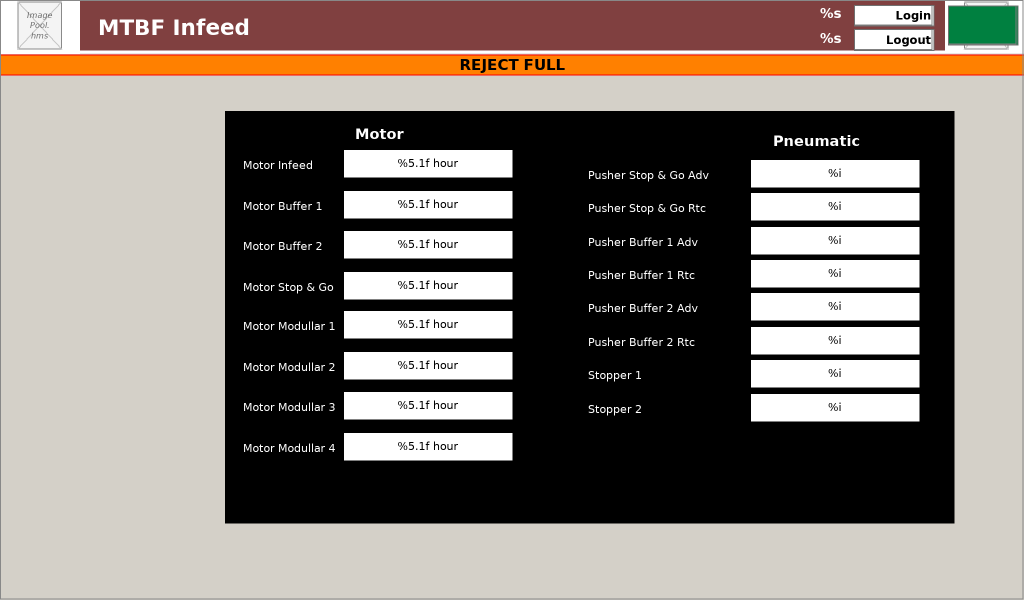
VISUALIZATION MTBF_Infeed  // 1024x600
    Frame (0,-2 1021x55)
        shows Header()
    Label (95,15 250x25), "MTBF Infeed"
    RoundedRectangle (225,111 729x412)
    Label (243,114 273x40), "Motor"
    Label (240,148 103x35), "Motor Infeed"
    RoundedRectangle (343,149 170x29), "%5.1f hour", text variable: InputOutput_GVL.MTBF_Motor[8]
    Label (240,189 103x35), "Motor Buffer 1"
    RoundedRectangle (343,190 170x29), "%5.1f hour", text variable: InputOutput_GVL.MTBF_Motor[9]
    Label (240,229 103x35), "Motor Buffer 2"
    RoundedRectangle (343,230 170x29), "%5.1f hour", text variable: InputOutput_GVL.MTBF_Motor[10]
    Label (240,270 103x35), "Motor Stop & Go"
    RoundedRectangle (343,271 170x29), "%5.1f hour", text variable: InputOutput_GVL.MTBF_Motor[11]
    Label (240,309 103x35), "Motor Modullar 1"
    RoundedRectangle (343,310 170x29), "%5.1f hour", text variable: InputOutput_GVL.MTBF_Motor[12]
    Label (240,350 103x35), "Motor Modullar 2"
    RoundedRectangle (343,351 170x29), "%5.1f hour", text variable: InputOutput_GVL.MTBF_Motor[13]
    Label (240,390 103x35), "Motor Modullar 3"
    RoundedRectangle (343,391 170x29), "%5.1f hour", text variable: InputOutput_GVL.MTBF_Motor[14]
    Label (240,431 103x35), "Motor Modullar 4"
    RoundedRectangle (343,432 170x29), "%5.1f hour", text variable: InputOutput_GVL.MTBF_Motor[15]
    Label (585,158 147x35), "Pusher Stop & Go Adv"
    RoundedRectangle (750,159 170x29), "%i", text variable: InputOutput_GVL.MTBF_Pneumatic[1]
    Label (680,121 273x40), "Pneumatic"
    Label (585,191 147x35), "Pusher Stop & Go Rtc"
    RoundedRectangle (750,192 170x29), "%i", text variable: InputOutput_GVL.MTBF_Pneumatic[2]
    Label (585,225 147x35), "Pusher Buffer 1 Adv"
    RoundedRectangle (750,226 170x29), "%i", text variable: InputOutput_GVL.MTBF_Pneumatic[3]
    Label (585,258 147x35), "Pusher Buffer 1 Rtc"
    RoundedRectangle (750,259 170x29), "%i", text variable: InputOutput_GVL.MTBF_Pneumatic[4]
    Label (585,291 147x35), "Pusher Buffer 2 Adv"
    RoundedRectangle (750,292 170x29), "%i", text variable: InputOutput_GVL.MTBF_Pneumatic[5]
    Label (585,325 147x35), "Pusher Buffer 2 Rtc"
    RoundedRectangle (750,326 170x29), "%i", text variable: InputOutput_GVL.MTBF_Pneumatic[6]
    Label (585,358 147x35), "Stopper 1"
    RoundedRectangle (750,359 170x29), "%i", text variable: InputOutput_GVL.MTBF_Pneumatic[7]
    Label (585,392 147x35), "Stopper 2"
    RoundedRectangle (750,393 170x29), "%i", text variable: InputOutput_GVL.MTBF_Pneumatic[8]
END_VISUALIZATION

// ---- VISUs/MTBF/MTBF_Shuttle.TcVIS
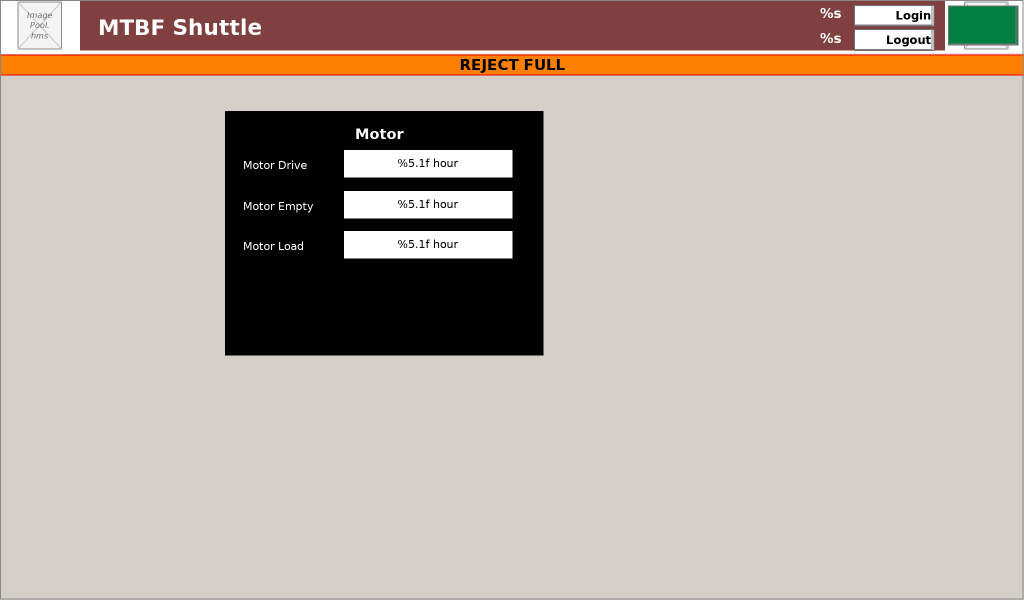
VISUALIZATION MTBF_Shuttle  // 1024x600
    Frame (0,-2 1021x55)
        shows Header()
    Label (95,15 250x25), "MTBF Shuttle"
    RoundedRectangle (225,111 318x244)
    Label (243,114 273x40), "Motor"
    Label (240,148 103x35), "Motor Drive"
    RoundedRectangle (343,149 170x29), "%5.1f hour", text variable: InputOutput_GVL.MTBF_Motor[16]
    Label (240,189 103x35), "Motor Empty"
    RoundedRectangle (343,190 170x29), "%5.1f hour", text variable: InputOutput_GVL.MTBF_Motor[17]
    Label (240,229 103x35), "Motor Load"
    RoundedRectangle (343,230 170x29), "%5.1f hour", text variable: InputOutput_GVL.MTBF_Motor[18]
END_VISUALIZATION

// ---- VISUs/MTBF/MTBF_Dispenser.TcVIS
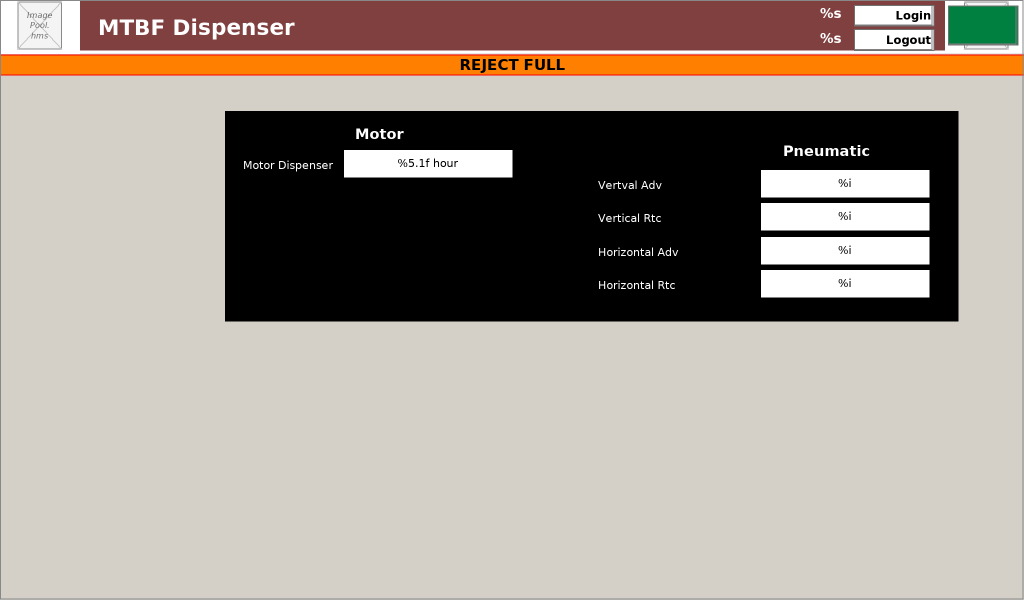
VISUALIZATION MTBF_Dispenser  // 1024x600
    Frame (0,-2 1021x55)
        shows Header()
    Label (95,15 250x25), "MTBF Dispenser"
    RoundedRectangle (225,111 733x210)
    Label (243,114 273x40), "Motor"
    Label (240,148 103x35), "Motor Dispenser"
    RoundedRectangle (343,149 170x29), "%5.1f hour", text variable: InputOutput_GVL.MTBF_Motor[19]
    Label (595,168 147x35), "Vertval Adv"
    RoundedRectangle (760,169 170x29), "%i", text variable: InputOutput_GVL.MTBF_Pneumatic[9]
    Label (690,131 273x40), "Pneumatic"
    Label (595,201 147x35), "Vertical Rtc"
    RoundedRectangle (760,202 170x29), "%i", text variable: InputOutput_GVL.MTBF_Pneumatic[10]
    Label (595,235 147x35), "Horizontal Adv"
    RoundedRectangle (760,236 170x29), "%i", text variable: InputOutput_GVL.MTBF_Pneumatic[11]
    Label (595,268 147x35), "Horizontal Rtc"
    RoundedRectangle (760,269 170x29), "%i", text variable: InputOutput_GVL.MTBF_Pneumatic[12]
END_VISUALIZATION

// ---- VISUs/OEE/OEE.TcVIS
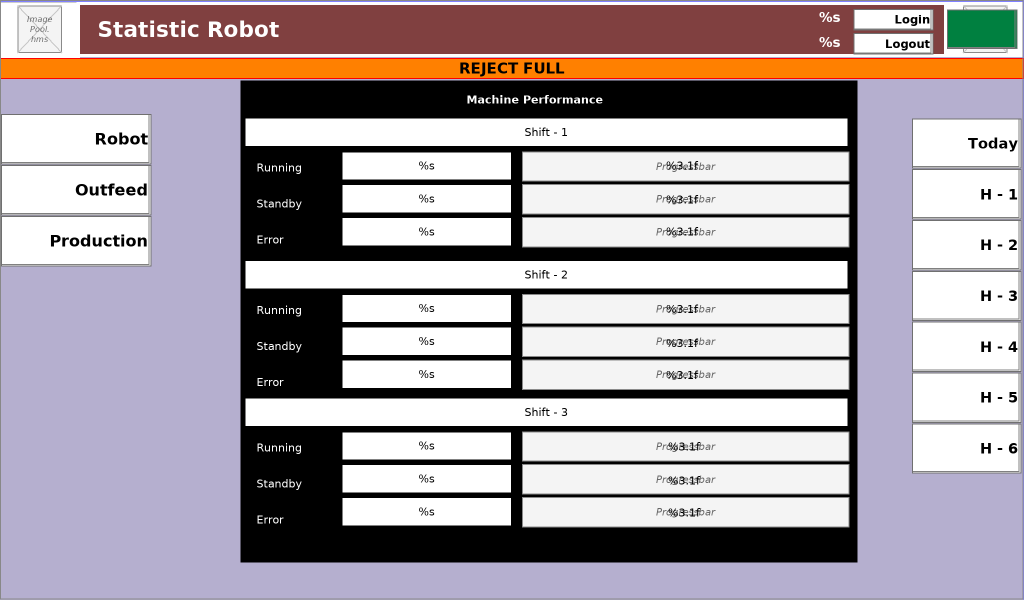
VISUALIZATION OEE  // 1024x600
    Frame (0,2 1023x598)
        shows OEE_Robot()
        shows OEE_Outfeed()
        shows OEE_Counter()
        shows Test_Place1()
        shows Test_Place2()
        shows Test_Place3()
        shows Test_Place4()
    Button (1,114 150x50), "Robot", image: VisuSymbols.Symbols.Database2
        OnMouseDown: FrameSelectionChange Selection=SelectedFrame=146e207b-fd78-4676-ba16-384fa245d7d2, GlobSel=AssignDir=MainPage.GenElemInst_1003, AssignType=Directly, SelType=Locally
    Button (1,165 150x50), "Outfeed", image: VisuSymbols.Symbols.Database2
        OnMouseDown: FrameSelectionChange Selection=SelectedFrame=146e207b-fd78-4676-ba16-384fa245d7d2, Selection=1, GlobSel=AssignDir=MainPage.GenElemInst_1003, AssignType=Directly, SelType=Locally
    Button (1,216 150x50), "Production", image: VisuSymbols.Symbols.Database2
        OnMouseDown: FrameSelectionChange Selection=SelectedFrame=146e207b-fd78-4676-ba16-384fa245d7d2, Selection=2, GlobSel=AssignDir=MainPage.GenElemInst_1003, AssignType=Directly, SelType=Locally
END_VISUALIZATION

// ---- VISUs/OEE/OEE_Outfeed.TcVIS
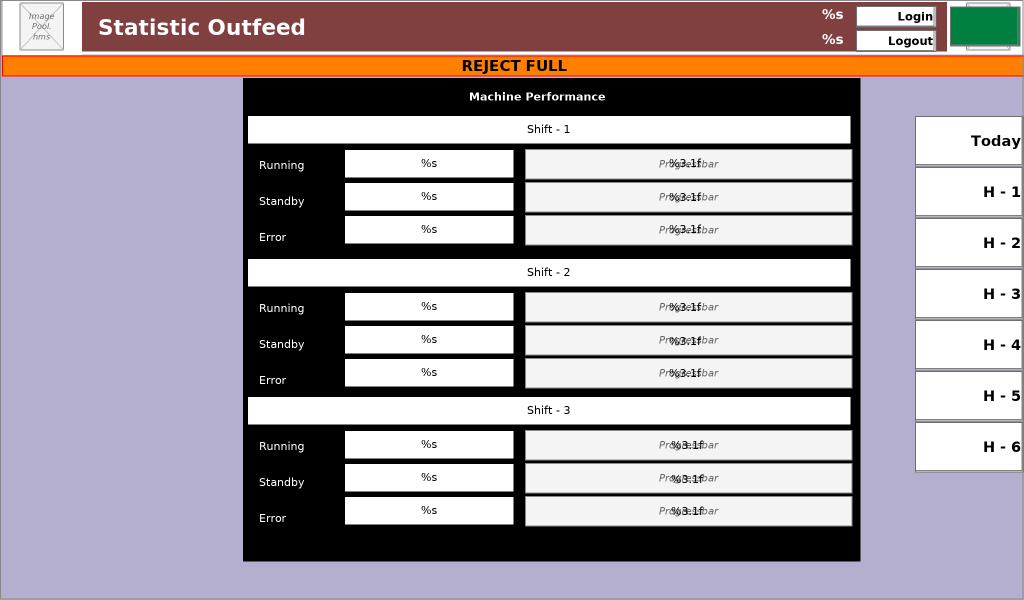
VISUALIZATION OEE_Outfeed  // 1024x600
    Frame (2,-1 1021x55)
        shows Header()
    RoundedRectangle (243,78 617x483)
    RoundedRectangle (247,115 604x29), "Shift - 1"
    Label (270,77 535x40), "Machine Performance"
    Label (256,148 78x35), "Running"
    Label (256,184 78x35), "Standby"
    Label (256,220 78x35), "Error"
    Progressbar (525,149 327x30), variable: Data_GVL.dt_OEEOutfeed.Precentage[0].Running
    Progressbar (525,182 327x30), variable: Data_GVL.dt_OEEOutfeed.Precentage[0].Stopped
    Progressbar (525,215 327x30), variable: Data_GVL.dt_OEEOutfeed.Precentage[0].Error
    RoundedRectangle (344,149 170x29), "%s", text variable: Data_GVL.dt_OEEOutfeed.HMI_Time[0].sRunning
    RoundedRectangle (344,182 170x29), "%s", text variable: Data_GVL.dt_OEEOutfeed.HMI_Time[0].sStopped
    RoundedRectangle (344,215 170x29), "%s", text variable: Data_GVL.dt_OEEOutfeed.HMI_Time[0].sError
    RoundedRectangle (247,258 604x29), "Shift - 2"
    Label (256,291 78x35), "Running"
    Label (256,327 78x35), "Standby"
    Label (256,363 78x35), "Error"
    Progressbar (525,292 327x30), variable: Data_GVL.dt_OEEOutfeed.Precentage[1].Running
    Progressbar (525,325 327x30), variable: Data_GVL.dt_OEEOutfeed.Precentage[1].Stopped
    Progressbar (525,358 327x30), variable: Data_GVL.dt_OEEOutfeed.Precentage[1].Error
    RoundedRectangle (344,292 170x29), "%s", text variable: Data_GVL.dt_OEEOutfeed.HMI_Time[1].sRunning
    RoundedRectangle (344,325 170x29), "%s", text variable: Data_GVL.dt_OEEOutfeed.HMI_Time[1].sStopped
    RoundedRectangle (344,358 170x29), "%s", text variable: Data_GVL.dt_OEEOutfeed.HMI_Time[1].sError
    RoundedRectangle (247,396 604x29), "Shift - 3"
    Label (256,429 78x35), "Running"
    Label (256,465 78x35), "Standby"
    Label (256,501 78x35), "Error"
    Progressbar (525,430 327x30), variable: Data_GVL.dt_OEEOutfeed.Precentage[2].Running
    Progressbar (525,463 327x30), variable: Data_GVL.dt_OEEOutfeed.Precentage[2].Stopped
    Progressbar (525,496 327x30), variable: Data_GVL.dt_OEEOutfeed.Precentage[2].Error
    RoundedRectangle (344,430 170x29), "%s", text variable: Data_GVL.dt_OEEOutfeed.HMI_Time[2].sRunning
    RoundedRectangle (344,463 170x29), "%s", text variable: Data_GVL.dt_OEEOutfeed.HMI_Time[2].sStopped
    RoundedRectangle (344,496 170x29), "%s", text variable: Data_GVL.dt_OEEOutfeed.HMI_Time[2].sError
    Button (915,116 109x50), "Today", image: VisuSymbols.Symbols.CalenderDay
        OnMouseClick: execute { Data_GVL.dt_OEEOutfeed.HMI_NumberPrev := 0; }
    Button (915,167 109x50), "H - 1", image: VisuSymbols.Symbols.CalenderDay
        OnMouseClick: execute { Data_GVL.dt_OEEOutfeed.HMI_NumberPrev := 1; }
    Button (915,218 109x50), "H - 2", image: VisuSymbols.Symbols.CalenderDay
        OnMouseClick: execute { Data_GVL.dt_OEEOutfeed.HMI_NumberPrev := 2; }
    Button (915,269 109x50), "H - 3", image: VisuSymbols.Symbols.CalenderDay
        OnMouseClick: execute { Data_GVL.dt_OEEOutfeed.HMI_NumberPrev := 3; }
    Button (915,320 109x50), "H - 4", image: VisuSymbols.Symbols.CalenderDay
        OnMouseClick: execute { Data_GVL.dt_OEEOutfeed.HMI_NumberPrev := 4; }
    Button (915,371 109x50), "H - 5", image: VisuSymbols.Symbols.CalenderDay
        OnMouseClick: execute { Data_GVL.dt_OEEOutfeed.HMI_NumberPrev := 5; }
    Button (915,422 109x50), "H - 6", image: VisuSymbols.Symbols.CalenderDay
        OnMouseClick: execute { Data_GVL.dt_OEEOutfeed.HMI_NumberPrev := 6; }
    RoundedRectangle (600,149 170x29), "%3.1f", text variable: Data_GVL.dt_OEEOutfeed.Precentage[0].Running
    RoundedRectangle (600,183 170x29), "%3.1f", text variable: Data_GVL.dt_OEEOutfeed.Precentage[0].Stopped
    RoundedRectangle (600,215 170x29), "%3.1f", text variable: Data_GVL.dt_OEEOutfeed.Precentage[0].Error
    RoundedRectangle (600,293 170x29), "%3.1f", text variable: Data_GVL.dt_OEEOutfeed.Precentage[1].Running
    RoundedRectangle (600,327 170x29), "%3.1f", text variable: Data_GVL.dt_OEEOutfeed.Precentage[1].Stopped
    RoundedRectangle (600,359 170x29), "%3.1f", text variable: Data_GVL.dt_OEEOutfeed.Precentage[1].Error
    RoundedRectangle (602,431 170x29), "%3.1f", text variable: Data_GVL.dt_OEEOutfeed.Precentage[2].Running
    RoundedRectangle (602,465 170x29), "%3.1f", text variable: Data_GVL.dt_OEEOutfeed.Precentage[2].Stopped
    RoundedRectangle (602,497 170x29), "%3.1f", text variable: Data_GVL.dt_OEEOutfeed.Precentage[2].Error
    Label (95,15 214x25), "Statistic Outfeed"
END_VISUALIZATION

// ---- VISUs/OEE/OEE_Robot.TcVIS
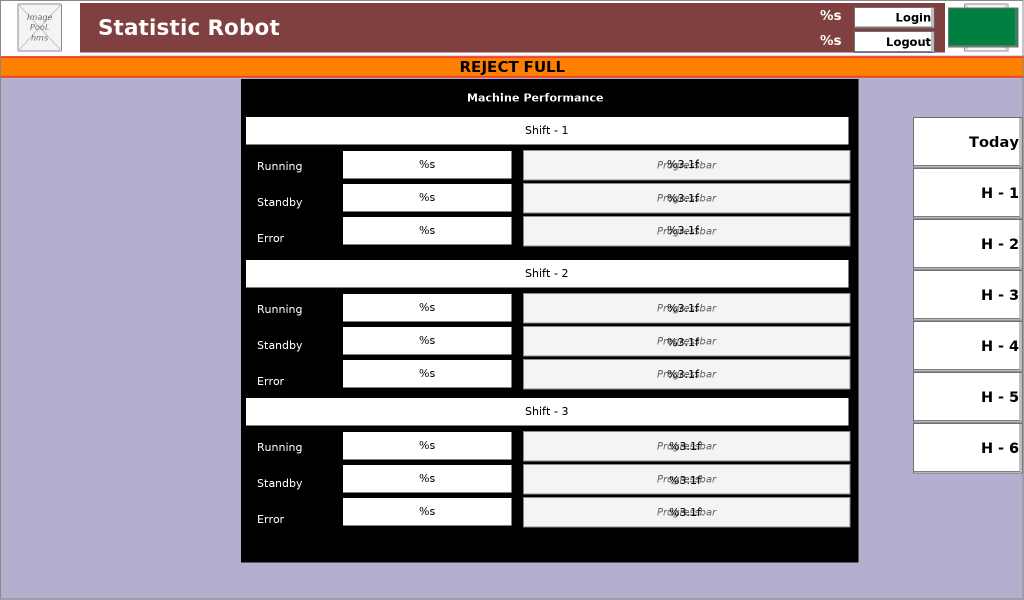
VISUALIZATION OEE_Robot  // 1024x600
    Frame (0,0 1021x55)
        shows Header()
    RoundedRectangle (241,79 617x483)
    RoundedRectangle (245,116 604x29), "Shift - 1"
    Label (268,78 535x40), "Machine Performance"
    Label (254,149 78x35), "Running"
    Label (254,185 78x35), "Standby"
    Label (254,221 78x35), "Error"
    Progressbar (523,150 327x30), variable: Data_GVL.dt_OEETime.Precentage[0].Running
    Progressbar (523,183 327x30), variable: Data_GVL.dt_OEETime.Precentage[0].Stopped
    Progressbar (523,216 327x30), variable: Data_GVL.dt_OEETime.Precentage[0].Error
    RoundedRectangle (342,150 170x29), "%s", text variable: Data_GVL.dt_OEETime.HMI_Time[0].sRunning
    RoundedRectangle (342,183 170x29), "%s", text variable: Data_GVL.dt_OEETime.HMI_Time[0].sStopped
    RoundedRectangle (342,216 170x29), "%s", text variable: Data_GVL.dt_OEETime.HMI_Time[0].sError
    RoundedRectangle (245,259 604x29), "Shift - 2"
    Label (254,292 78x35), "Running"
    Label (254,328 78x35), "Standby"
    Label (254,364 78x35), "Error"
    Progressbar (523,293 327x30), variable: Data_GVL.dt_OEETime.Precentage[1].Running
    Progressbar (523,326 327x30), variable: Data_GVL.dt_OEETime.Precentage[1].Stopped
    Progressbar (523,359 327x30), variable: Data_GVL.dt_OEETime.Precentage[1].Error
    RoundedRectangle (342,293 170x29), "%s", text variable: Data_GVL.dt_OEETime.HMI_Time[1].sRunning
    RoundedRectangle (342,326 170x29), "%s", text variable: Data_GVL.dt_OEETime.HMI_Time[1].sStopped
    RoundedRectangle (342,359 170x29), "%s", text variable: Data_GVL.dt_OEETime.HMI_Time[1].sError
    RoundedRectangle (245,397 604x29), "Shift - 3"
    Label (254,430 78x35), "Running"
    Label (254,466 78x35), "Standby"
    Label (254,502 78x35), "Error"
    Progressbar (523,431 327x30), variable: Data_GVL.dt_OEETime.Precentage[2].Running
    Progressbar (523,464 327x30), variable: Data_GVL.dt_OEETime.Precentage[2].Stopped
    Progressbar (523,497 327x30), variable: Data_GVL.dt_OEETime.Precentage[2].Error
    RoundedRectangle (342,431 170x29), "%s", text variable: Data_GVL.dt_OEETime.HMI_Time[2].sRunning
    RoundedRectangle (342,464 170x29), "%s", text variable: Data_GVL.dt_OEETime.HMI_Time[2].sStopped
    RoundedRectangle (342,497 170x29), "%s", text variable: Data_GVL.dt_OEETime.HMI_Time[2].sError
    Button (913,117 109x50), "Today", image: VisuSymbols.Symbols.CalenderDay
        OnMouseClick: execute { Data_GVL.dt_OEETime.HMI_NumberPrev := 0; }
    Button (913,168 109x50), "H - 1", image: VisuSymbols.Symbols.CalenderDay
        OnMouseClick: execute { Data_GVL.dt_OEETime.HMI_NumberPrev := 1; }
    Button (913,219 109x50), "H - 2", image: VisuSymbols.Symbols.CalenderDay
        OnMouseClick: execute { Data_GVL.dt_OEETime.HMI_NumberPrev := 2; }
    Button (913,270 109x50), "H - 3", image: VisuSymbols.Symbols.CalenderDay
        OnMouseClick: execute { Data_GVL.dt_OEETime.HMI_NumberPrev := 3; }
    Button (913,321 109x50), "H - 4", image: VisuSymbols.Symbols.CalenderDay
        OnMouseClick: execute { Data_GVL.dt_OEETime.HMI_NumberPrev := 4; }
    Button (913,372 109x50), "H - 5", image: VisuSymbols.Symbols.CalenderDay
        OnMouseClick: execute { Data_GVL.dt_OEETime.HMI_NumberPrev := 5; }
    Button (913,423 109x50), "H - 6", image: VisuSymbols.Symbols.CalenderDay
        OnMouseClick: execute { Data_GVL.dt_OEETime.HMI_NumberPrev := 6; }
    RoundedRectangle (598,150 170x29), "%3.1f", text variable: Data_GVL.dt_OEETime.Precentage[0].Running
    RoundedRectangle (598,184 170x29), "%3.1f", text variable: Data_GVL.dt_OEETime.Precentage[0].Stopped
    RoundedRectangle (598,216 170x29), "%3.1f", text variable: Data_GVL.dt_OEETime.Precentage[0].Error
    RoundedRectangle (598,294 170x29), "%3.1f", text variable: Data_GVL.dt_OEETime.Precentage[1].Running
    RoundedRectangle (598,328 170x29), "%3.1f", text variable: Data_GVL.dt_OEETime.Precentage[1].Stopped
    RoundedRectangle (598,360 170x29), "%3.1f", text variable: Data_GVL.dt_OEETime.Precentage[1].Error
    RoundedRectangle (600,432 170x29), "%3.1f", text variable: Data_GVL.dt_OEETime.Precentage[2].Running
    RoundedRectangle (600,466 170x29), "%3.1f", text variable: Data_GVL.dt_OEETime.Precentage[2].Stopped
    RoundedRectangle (600,498 170x29), "%3.1f", text variable: Data_GVL.dt_OEETime.Precentage[2].Error
    Label (95,15 214x25), "Statistic Robot"
END_VISUALIZATION

// ---- VISUs/OEE/OEE_Counter.TcVIS
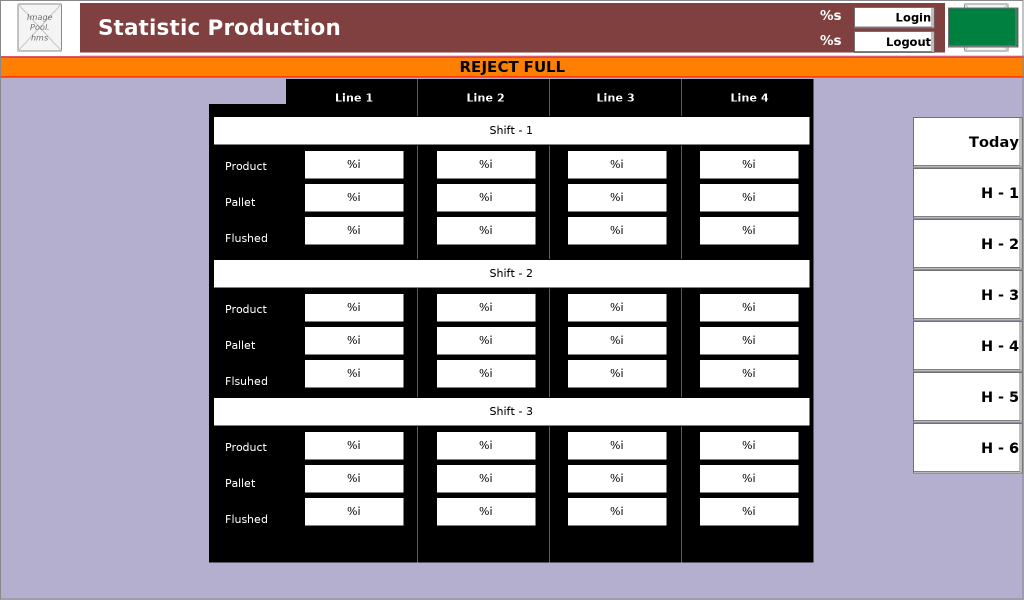
VISUALIZATION OEE_Counter  // 1024x600
    Frame (0,0 1021x55)
        shows Header()
    Button (913,117 109x50), "Today", image: VisuSymbols.Symbols.CalenderDay
        OnMouseClick: execute {
            Data_GVL.dt_OEECounter[1].HMI_NumberPrev := 0;
            Data_GVL.dt_OEECounter[2].HMI_NumberPrev := 0;
            Data_GVL.dt_OEECounter[3].HMI_NumberPrev := 0;
            Data_GVL.dt_OEECounter[4].HMI_NumberPrev := 0;
        }
    Button (913,168 109x50), "H - 1", image: VisuSymbols.Symbols.CalenderDay
        OnMouseClick: execute {
            Data_GVL.dt_OEECounter[1].HMI_NumberPrev := 1;
            Data_GVL.dt_OEECounter[2].HMI_NumberPrev := 1;
            Data_GVL.dt_OEECounter[3].HMI_NumberPrev := 1;
            Data_GVL.dt_OEECounter[4].HMI_NumberPrev := 1;
        }
    Button (913,219 109x50), "H - 2", image: VisuSymbols.Symbols.CalenderDay
        OnMouseClick: execute {
            Data_GVL.dt_OEECounter[1].HMI_NumberPrev := 2;
            Data_GVL.dt_OEECounter[2].HMI_NumberPrev := 2;
            Data_GVL.dt_OEECounter[3].HMI_NumberPrev := 2;
            Data_GVL.dt_OEECounter[4].HMI_NumberPrev := 2;
        }
    Button (913,270 109x50), "H - 3", image: VisuSymbols.Symbols.CalenderDay
        OnMouseClick: execute {
            Data_GVL.dt_OEECounter[1].HMI_NumberPrev := 3;
            Data_GVL.dt_OEECounter[2].HMI_NumberPrev := 3;
            Data_GVL.dt_OEECounter[3].HMI_NumberPrev := 3;
            Data_GVL.dt_OEECounter[4].HMI_NumberPrev := 3;
        }
    Button (913,321 109x50), "H - 4", image: VisuSymbols.Symbols.CalenderDay
        OnMouseClick: execute {
            Data_GVL.dt_OEECounter[1].HMI_NumberPrev := 4;
            Data_GVL.dt_OEECounter[2].HMI_NumberPrev := 4;
            Data_GVL.dt_OEECounter[3].HMI_NumberPrev := 4;
            Data_GVL.dt_OEECounter[4].HMI_NumberPrev := 4;
        }
    Button (913,372 109x50), "H - 5", image: VisuSymbols.Symbols.CalenderDay
        OnMouseClick: execute {
            Data_GVL.dt_OEECounter[1].HMI_NumberPrev := 5;
            Data_GVL.dt_OEECounter[2].HMI_NumberPrev := 5;
            Data_GVL.dt_OEECounter[3].HMI_NumberPrev := 5;
            Data_GVL.dt_OEECounter[4].HMI_NumberPrev := 5;
        }
    Button (913,423 109x50), "H - 6", image: VisuSymbols.Symbols.CalenderDay
        OnMouseClick: execute {
            Data_GVL.dt_OEECounter[1].HMI_NumberPrev := 6;
            Data_GVL.dt_OEECounter[2].HMI_NumberPrev := 6;
            Data_GVL.dt_OEECounter[3].HMI_NumberPrev := 6;
            Data_GVL.dt_OEECounter[4].HMI_NumberPrev := 6;
        }
    Label (95,15 240x25), "Statistic Production"
    RoundedRectangle (286,79 131x483)
    RoundedRectangle (418,79 131x483)
    RoundedRectangle (682,79 131x483)
    RoundedRectangle (550,79 131x483)
    RoundedRectangle (209,104 207x458)
    RoundedRectangle (213,116 597x29), "Shift - 1"
    Label (312,78 84x40), "Line 1"
    Label (222,149 78x35), "Product"
    Label (222,185 78x35), "Pallet"
    Label (222,221 78x35), "Flushed"
    RoundedRectangle (304,150 100x29), "%i", text variable: Data_GVL.dt_OEECounter[1].HMI_Counter[0].Data1
    RoundedRectangle (304,183 100x29), "%i", text variable: Data_GVL.dt_OEECounter[1].HMI_Counter[0].Data2
    RoundedRectangle (304,216 100x29), "%i", text variable: Data_GVL.dt_OEECounter[1].HMI_Counter[0].Data3
    RoundedRectangle (213,259 597x29), "Shift - 2"
    Label (222,292 78x35), "Product"
    Label (222,328 78x35), "Pallet"
    Label (222,364 78x35), "Flsuhed"
    RoundedRectangle (304,293 100x29), "%i", text variable: Data_GVL.dt_OEECounter[1].HMI_Counter[1].Data1
    RoundedRectangle (304,326 100x29), "%i", text variable: Data_GVL.dt_OEECounter[1].HMI_Counter[1].Data2
    RoundedRectangle (304,359 100x29), "%i", text variable: Data_GVL.dt_OEECounter[1].HMI_Counter[1].Data3
    RoundedRectangle (213,397 597x29), "Shift - 3"
    Label (222,430 78x35), "Product"
    Label (222,466 78x35), "Pallet"
    Label (222,502 78x35), "Flushed"
    RoundedRectangle (304,431 100x29), "%i", text variable: Data_GVL.dt_OEECounter[1].HMI_Counter[2].Data1
    RoundedRectangle (304,464 100x29), "%i", text variable: Data_GVL.dt_OEECounter[1].HMI_Counter[2].Data2
    RoundedRectangle (304,497 100x29), "%i", text variable: Data_GVL.dt_OEECounter[1].HMI_Counter[2].Data3
    Label (438,78 95x40), "Line 2"
    RoundedRectangle (436,150 100x29), "%i", text variable: Data_GVL.dt_OEECounter[2].HMI_Counter[0].Data1
    RoundedRectangle (436,183 100x29), "%i", text variable: Data_GVL.dt_OEECounter[2].HMI_Counter[0].Data2
    RoundedRectangle (436,216 100x29), "%i", text variable: Data_GVL.dt_OEECounter[2].HMI_Counter[0].Data3
    RoundedRectangle (436,293 100x29), "%i", text variable: Data_GVL.dt_OEECounter[2].HMI_Counter[1].Data1
    RoundedRectangle (436,326 100x29), "%i", text variable: Data_GVL.dt_OEECounter[2].HMI_Counter[1].Data2
    RoundedRectangle (436,359 100x29), "%i", text variable: Data_GVL.dt_OEECounter[2].HMI_Counter[1].Data3
    RoundedRectangle (436,431 100x29), "%i", text variable: Data_GVL.dt_OEECounter[2].HMI_Counter[2].Data1
    RoundedRectangle (436,464 100x29), "%i", text variable: Data_GVL.dt_OEECounter[2].HMI_Counter[2].Data2
    RoundedRectangle (436,497 100x29), "%i", text variable: Data_GVL.dt_OEECounter[2].HMI_Counter[2].Data3
    RoundedRectangle (567,150 100x29), "%i", text variable: Data_GVL.dt_OEECounter[3].HMI_Counter[0].Data1
    RoundedRectangle (567,183 100x29), "%i", text variable: Data_GVL.dt_OEECounter[3].HMI_Counter[0].Data2
    RoundedRectangle (567,216 100x29), "%i", text variable: Data_GVL.dt_OEECounter[3].HMI_Counter[0].Data3
    RoundedRectangle (567,293 100x29), "%i", text variable: Data_GVL.dt_OEECounter[3].HMI_Counter[1].Data1
    RoundedRectangle (567,326 100x29), "%i", text variable: Data_GVL.dt_OEECounter[3].HMI_Counter[1].Data2
    RoundedRectangle (567,359 100x29), "%i", text variable: Data_GVL.dt_OEECounter[3].HMI_Counter[1].Data3
    RoundedRectangle (567,431 100x29), "%i", text variable: Data_GVL.dt_OEECounter[3].HMI_Counter[2].Data1
    RoundedRectangle (567,464 100x29), "%i", text variable: Data_GVL.dt_OEECounter[3].HMI_Counter[2].Data2
    RoundedRectangle (567,497 100x29), "%i", text variable: Data_GVL.dt_OEECounter[3].HMI_Counter[2].Data3
    RoundedRectangle (699,150 100x29), "%i", text variable: Data_GVL.dt_OEECounter[4].HMI_Counter[0].Data1
    RoundedRectangle (699,183 100x29), "%i", text variable: Data_GVL.dt_OEECounter[4].HMI_Counter[0].Data2
    RoundedRectangle (699,216 100x29), "%i", text variable: Data_GVL.dt_OEECounter[4].HMI_Counter[0].Data3
    RoundedRectangle (699,293 100x29), "%i", text variable: Data_GVL.dt_OEECounter[4].HMI_Counter[1].Data1
    RoundedRectangle (699,326 100x29), "%i", text variable: Data_GVL.dt_OEECounter[4].HMI_Counter[1].Data2
    RoundedRectangle (699,359 100x29), "%i", text variable: Data_GVL.dt_OEECounter[4].HMI_Counter[1].Data3
    RoundedRectangle (699,431 100x29), "%i", text variable: Data_GVL.dt_OEECounter[4].HMI_Counter[2].Data1
    RoundedRectangle (699,464 100x29), "%i", text variable: Data_GVL.dt_OEECounter[4].HMI_Counter[2].Data2
    RoundedRectangle (699,497 100x29), "%i", text variable: Data_GVL.dt_OEECounter[4].HMI_Counter[2].Data3
    Label (568,78 95x40), "Line 3"
    Label (702,78 95x40), "Line 4"
END_VISUALIZATION

// ---- VISUs/Parameter/LinkUp.TcTLO
TEXTLIST LinkUp
  1 = 'LU 11'
  2 = 'LU 12'
  3 = 'LU 13'
  4 = 'LU 14'
  5 = 'LU 16'
  6 = 'LU 17'
  7 = 'LU 18'
  8 = 'LU 21'
  9 = 'LU 22'
  10 = 'LU 23'
  11 = 'LU 24'
  12 = 'LU 26'
  13 = 'LU 27'
  14 = 'LU 29'
   = ''
END_TEXTLIST

// ---- VISUs/Parameter/MShuttle.TcVIS
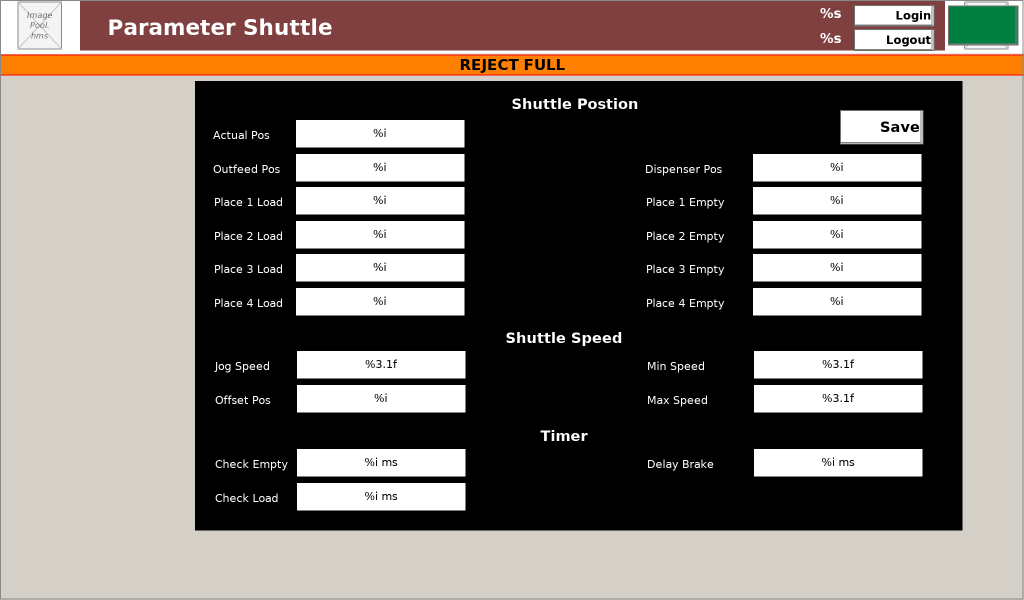
VISUALIZATION MShuttle  // 1024x600
    Frame (0,-2 1021x55)
        shows Header()
    Label (95,15 250x25), "Parameter Shuttle"
    RoundedRectangle (195,81 767x449)
    Label (223,84 704x40), "Shuttle Postion"
    Label (210,118 78x35), "Actual Pos"
    RoundedRectangle (295,119 170x29), "%i", text variable: InputOutput_GVL.ShuttlePosition
    Button (840,110 83x34), "Save", image: VisuSymbols.Symbols.Save
        tap InputOutput_GVL.TestMode[100]
    Label (210,152 78x35), "Outfeed Pos"
    RoundedRectangle (295,153 170x29), "%i", text variable: HMI_GVL.stShuttleSequence[0].PositionLoaded
        OnMouseClick: write the text variable via Default
    Label (642,152 102x35), "Dispenser Pos"
    RoundedRectangle (752,153 170x29), "%i", text variable: HMI_GVL.stShuttleSequence[0].PositionEmpty
        OnMouseClick: write the text variable via Default
    Label (211,185 78x35), "Place 1 Load"
    RoundedRectangle (295,186 170x29), "%i", text variable: HMI_GVL.stShuttleSequence[1].PositionLoaded
        OnMouseClick: write the text variable via Default
    Label (643,185 102x35), "Place 1 Empty"
    RoundedRectangle (752,186 170x29), "%i", text variable: HMI_GVL.stShuttleSequence[1].PositionEmpty
        OnMouseClick: write the text variable via Default
    Label (211,219 78x35), "Place 2 Load"
    RoundedRectangle (295,220 170x29), "%i", text variable: HMI_GVL.stShuttleSequence[2].PositionLoaded
        OnMouseClick: write the text variable via Default
    Label (643,219 102x35), "Place 2 Empty"
    RoundedRectangle (752,220 170x29), "%i", text variable: HMI_GVL.stShuttleSequence[2].PositionEmpty
        OnMouseClick: write the text variable via Default
    Label (211,252 78x35), "Place 3 Load"
    RoundedRectangle (295,253 170x29), "%i", text variable: HMI_GVL.stShuttleSequence[3].PositionLoaded
        OnMouseClick: write the text variable via Default
    Label (643,252 102x35), "Place 3 Empty"
    RoundedRectangle (752,253 170x29), "%i", text variable: HMI_GVL.stShuttleSequence[3].PositionEmpty
        OnMouseClick: write the text variable via Default
    Label (211,286 78x35), "Place 4 Load"
    RoundedRectangle (295,287 170x29), "%i", text variable: HMI_GVL.stShuttleSequence[4].PositionLoaded
        OnMouseClick: write the text variable via Default
    Label (643,286 102x35), "Place 4 Empty"
    RoundedRectangle (752,287 170x29), "%i", text variable: HMI_GVL.stShuttleSequence[4].PositionEmpty
        OnMouseClick: write the text variable via Default
    Label (212,318 704x40), "Shuttle Speed"
    Label (212,349 78x35), "Jog Speed"
    RoundedRectangle (296,350 170x29), "%3.1f", text variable: HMI_GVL.Shuttle_JogSpeed
        OnMouseClick: write the text variable via Default
    Label (644,349 102x35), "Min Speed"
    RoundedRectangle (753,350 170x29), "%3.1f", text variable: HMI_GVL.Shuttle_MinSpeed
        OnMouseClick: write the text variable via Default
    Label (212,383 78x35), "Offset Pos"
    RoundedRectangle (296,384 170x29), "%i", text variable: HMI_GVL.Shuttle_Offset
        OnMouseClick: write the text variable via Default
    Label (644,383 102x35), "Max Speed"
    RoundedRectangle (753,384 170x29), "%3.1f", text variable: HMI_GVL.Shuttle_MaxSpeed
        OnMouseClick: write the text variable via Default
    Label (212,416 704x40), "Timer"
    Label (212,447 78x35), "Check Empty"
    RoundedRectangle (296,448 170x29), "%i ms", text variable: HMI_GVL.Tmr_EmptyShuttle
        OnMouseClick: write the text variable via Default
    Label (644,447 102x35), "Delay Brake"
    RoundedRectangle (753,448 170x29), "%i ms", text variable: HMI_GVL.Tmr_BrakeShuttle
        OnMouseClick: write the text variable via Default
    Label (212,481 78x35), "Check Load"
    RoundedRectangle (296,482 170x29), "%i ms", text variable: HMI_GVL.Tmr_LoadedShuttle
        OnMouseClick: write the text variable via Default
END_VISUALIZATION

// ---- VISUs/Parameter/MOutfeed.TcVIS
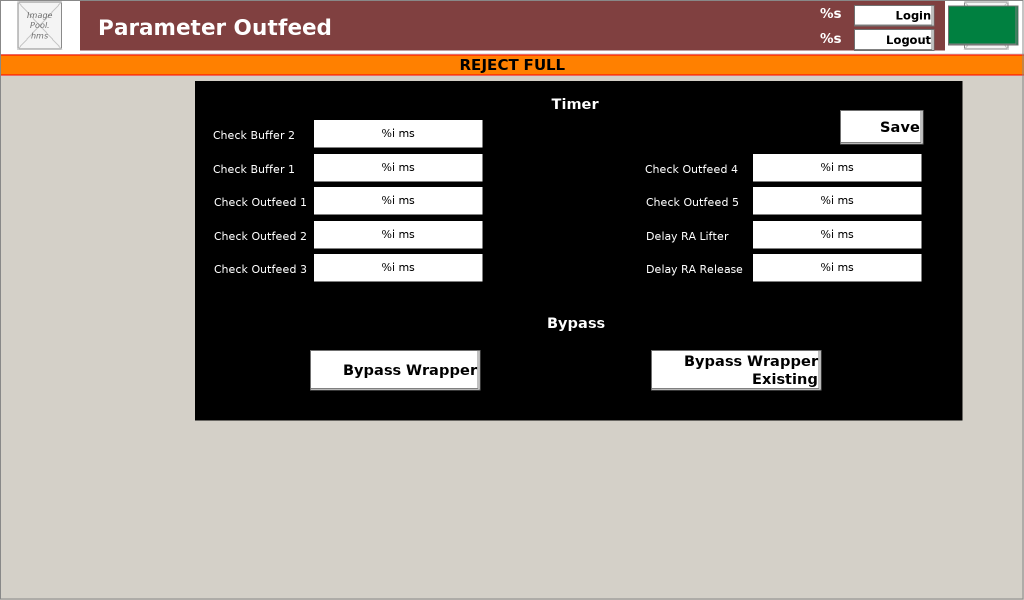
VISUALIZATION MOutfeed  // 1024x600
    Frame (0,-2 1021x55)
        shows Header()
    Label (95,15 250x25), "Parameter Outfeed"
    RoundedRectangle (195,81 767x339)
    Label (223,84 704x40), "Timer"
    Label (210,118 91x35), "Check Buffer 2"
    RoundedRectangle (313,119 170x29), "%i ms", text variable: HMI_GVL.Tmr_PalletBuffer2
        OnMouseClick: write the text variable via Default
    Button (840,110 83x34), "Save", image: VisuSymbols.Symbols.Save
        tap InputOutput_GVL.TestMode[100]
    Label (210,152 91x35), "Check Buffer 1"
    RoundedRectangle (313,153 170x29), "%i ms", text variable: HMI_GVL.Tmr_PalletBuffer1
        OnMouseClick: write the text variable via Default
    Label (642,152 102x35), "Check Outfeed 4"
    RoundedRectangle (752,153 170x29), "%i ms", text variable: HMI_GVL.Tmr_PalletOutfeed4
        OnMouseClick: write the text variable via Default
    Label (211,185 102x35), "Check Outfeed 1"
    RoundedRectangle (313,186 170x29), "%i ms", text variable: HMI_GVL.Tmr_PalletOutfeed1
        OnMouseClick: write the text variable via Default
    Label (643,185 102x35), "Check Outfeed 5"
    RoundedRectangle (752,186 170x29), "%i ms", text variable: HMI_GVL.Tmr_PalletOutfeed5
        OnMouseClick: write the text variable via Default
    Label (211,219 100x35), "Check Outfeed 2"
    RoundedRectangle (313,220 170x29), "%i ms", text variable: HMI_GVL.Tmr_PalletOutfeed2
        OnMouseClick: write the text variable via Default
    Label (643,219 102x35), "Delay RA Lifter"
    RoundedRectangle (752,220 170x29), "%i ms", text variable: HMI_GVL.Tmr_PalletRA
        OnMouseClick: write the text variable via Default
    Label (211,252 100x35), "Check Outfeed 3"
    RoundedRectangle (313,253 170x29), "%i ms", text variable: HMI_GVL.Tmr_PalletOutfeed3
        OnMouseClick: write the text variable via Default
    Label (643,252 102x35), "Delay RA Release"
    RoundedRectangle (752,253 170x29), "%i ms", text variable: HMI_GVL.TmrDelay_PalletRA
        OnMouseClick: write the text variable via Default
    Label (224,303 704x40), "Bypass"
    Button (651,350 170x40), "Bypass Wrapper Existing", colour toggle: HMI_GVL.BypassWrapperExisting, image: VisuSymbols.Symbols.Lock
        toggle HMI_GVL.BypassWrapperExisting
    Button (310,350 170x40), "Bypass Wrapper", colour toggle: HMI_GVL.BypassWrapper, image: VisuSymbols.Symbols.Lock
        toggle HMI_GVL.BypassWrapper
END_VISUALIZATION

// ---- VISUs/Parameter/MInfeed.TcVIS
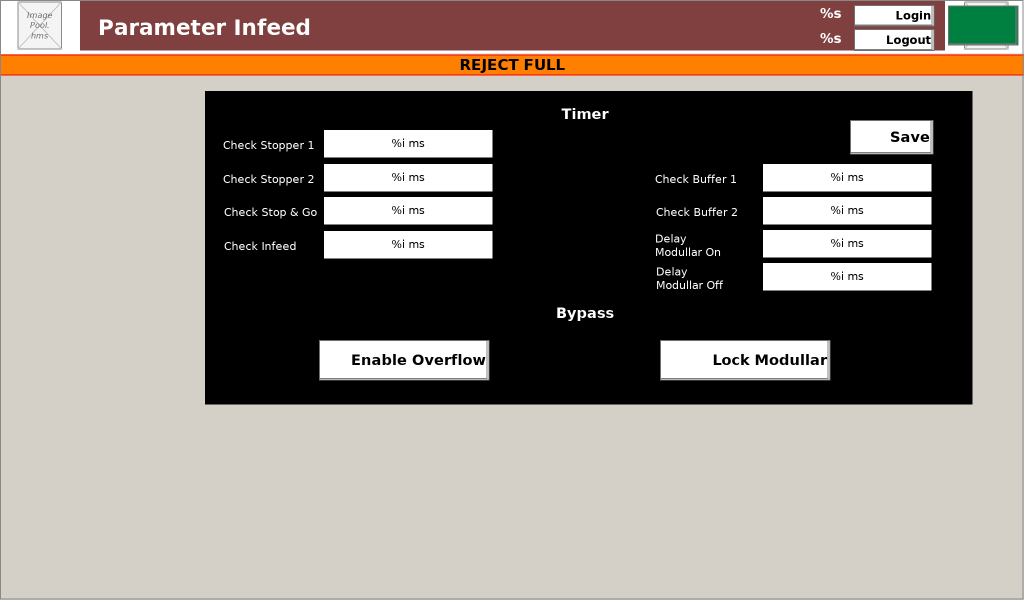
VISUALIZATION MInfeed  // 1024x600
    Frame (0,-2 1021x55)
        shows Header()
    Label (95,15 250x25), "Parameter Infeed"
    RoundedRectangle (205,91 767x313)
    Label (233,94 704x40), "Timer"
    Label (220,128 103x35), "Check Stopper 1"
    RoundedRectangle (323,129 170x29), "%i ms", text variable: HMI_GVL.Tmr_Stopper1
        OnMouseClick: write the text variable via Default
    Button (850,120 83x34), "Save", image: VisuSymbols.Symbols.Save
        tap InputOutput_GVL.TestMode[100]
    Label (220,162 104x35), "Check Stopper 2"
    RoundedRectangle (323,163 170x29), "%i ms", text variable: HMI_GVL.Tmr_Stopper2
        OnMouseClick: write the text variable via Default
    Label (652,162 102x35), "Check Buffer 1"
    RoundedRectangle (762,163 170x29), "%i ms", text variable: HMI_GVL.Tmr_Buffer1
        OnMouseClick: write the text variable via Default
    Label (221,195 102x35), "Check Stop & Go"
    RoundedRectangle (323,196 170x29), "%i ms", text variable: HMI_GVL.Tmr_StopGo
        OnMouseClick: write the text variable via Default
    Label (653,195 102x35), "Check Buffer 2"
    RoundedRectangle (762,196 170x29), "%i ms", text variable: HMI_GVL.Tmr_Buffer2
        OnMouseClick: write the text variable via Default
    Label (221,229 100x35), "Check Infeed"
    RoundedRectangle (323,230 170x29), "%i ms", text variable: HMI_GVL.Tmr_Infeed
        OnMouseClick: write the text variable via Default
    Label (233,293 704x40), "Bypass"
    Button (660,340 170x40), "Lock Modullar", colour toggle: HMI_GVL.LockModullarToRun, image: VisuSymbols.Symbols.Lock
        toggle HMI_GVL.LockModullarToRun
    Label (652,228 102x35), "Delay Modullar On"
    RoundedRectangle (762,229 170x29), "%i ms", text variable: HMI_GVL.Tmr_ModullarOn
        OnMouseClick: write the text variable via Default
    Label (653,261 102x35), "Delay Modullar Off"
    RoundedRectangle (762,262 170x29), "%i ms", text variable: HMI_GVL.Tmr_ModullarOff
        OnMouseClick: write the text variable via Default
    Button (319,340 170x40), "Enable Overflow", colour toggle: HMI_GVL.Disable_Overflow, image: VisuSymbols.Symbols.Lock
        toggle HMI_GVL.Disable_Overflow
END_VISUALIZATION

// ---- VISUs/Parameter/MDispenser.TcVIS
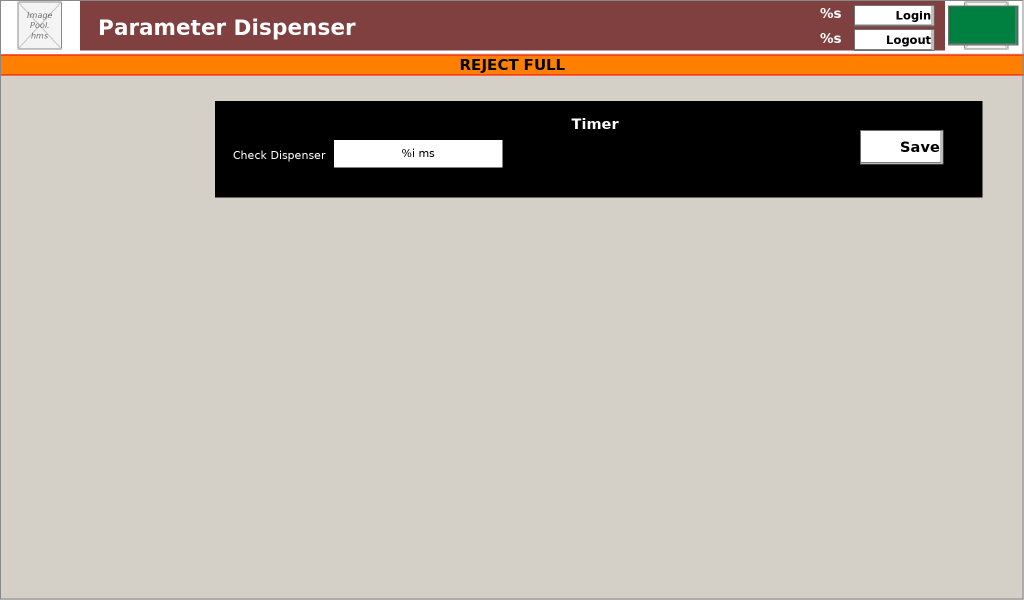
VISUALIZATION MDispenser  // 1024x600
    Frame (0,-2 1021x55)
        shows Header()
    Label (95,15 250x25), "Parameter Dispenser"
    RoundedRectangle (215,101 767x96)
    Label (243,104 704x40), "Timer"
    Label (230,138 103x35), "Check Dispenser"
    RoundedRectangle (333,139 170x29), "%i ms", text variable: HMI_GVL.Tmr_Dispenser
        OnMouseClick: write the text variable via Default
    Button (860,130 83x34), "Save", image: VisuSymbols.Symbols.Save
        tap InputOutput_GVL.TestMode[100]
END_VISUALIZATION

// ---- VISUs/Parameter/MPicking.TcVIS
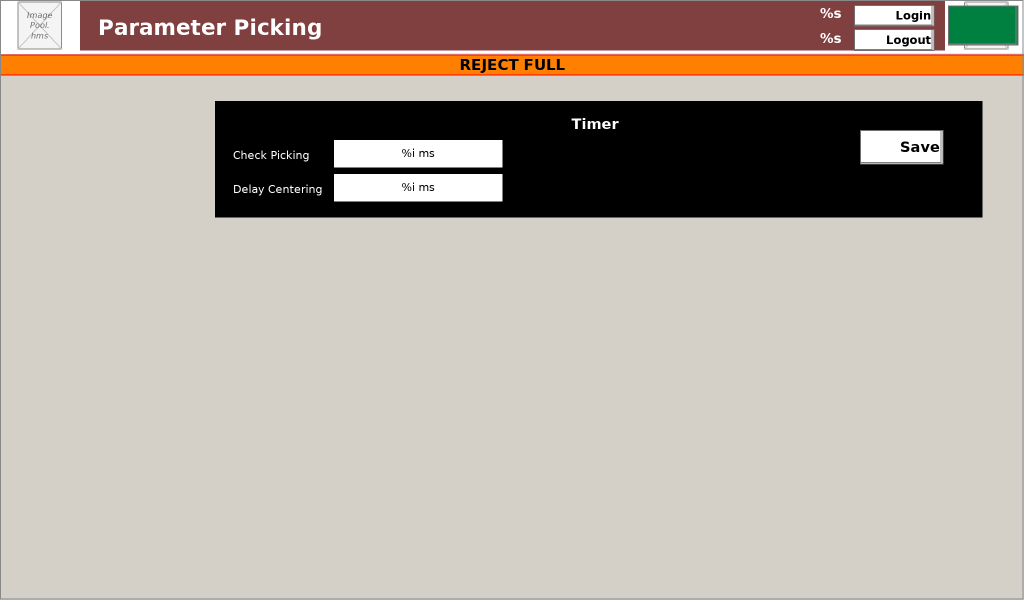
VISUALIZATION MPicking  // 1024x600
    Frame (0,-2 1021x55)
        shows Header()
    Label (95,15 250x25), "Parameter Picking"
    RoundedRectangle (215,101 767x116)
    Label (243,104 704x40), "Timer"
    Label (230,138 103x35), "Check Picking"
    RoundedRectangle (333,139 170x29), "%i ms", text variable: HMI_GVL.Tmr_Picking
        OnMouseClick: write the text variable via Default
    Button (860,130 83x34), "Save", image: VisuSymbols.Symbols.Save
        tap InputOutput_GVL.TestMode[100]
    Label (230,172 104x35), "Delay Centering"
    RoundedRectangle (333,173 170x29), "%i ms", text variable: HMI_GVL.Tmr_Centering
        OnMouseClick: write the text variable via Default
END_VISUALIZATION

// ---- VISUs/Parameter/MPlacing.TcVIS
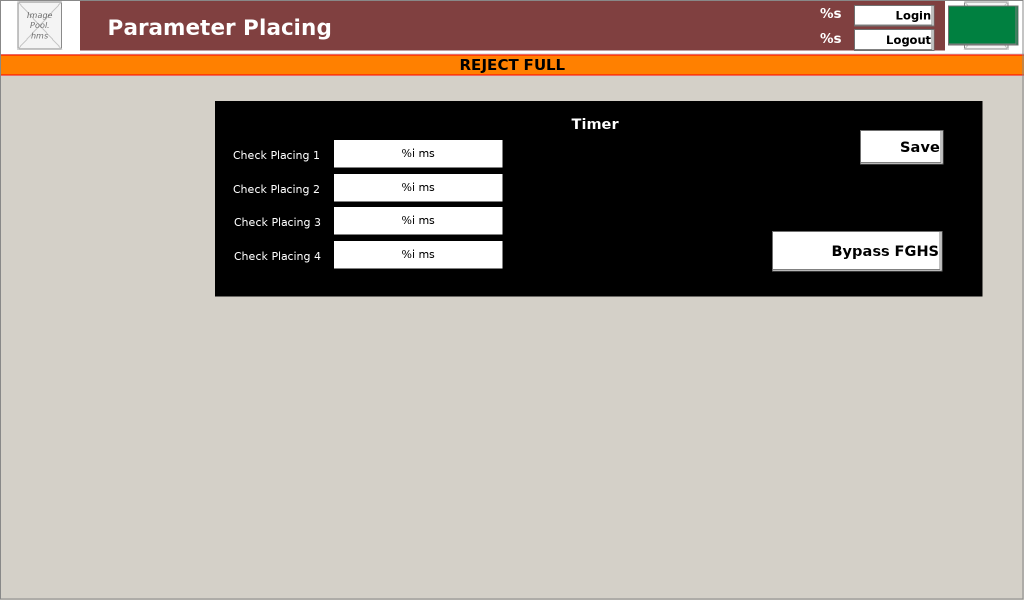
VISUALIZATION MPlacing  // 1024x600
    Frame (0,-2 1021x55)
        shows Header()
    Label (95,15 250x25), "Parameter Placing"
    RoundedRectangle (215,101 767x195)
    Label (243,104 704x40), "Timer"
    Label (230,138 103x35), "Check Placing 1"
    RoundedRectangle (333,139 170x29), "%i ms", text variable: HMI_GVL.Tmr_Placing1
        OnMouseClick: write the text variable via Default
    Button (860,130 83x34), "Save", image: VisuSymbols.Symbols.Save
        tap InputOutput_GVL.TestMode[100]
    Label (230,172 104x35), "Check Placing 2"
    RoundedRectangle (333,173 170x29), "%i ms", text variable: HMI_GVL.Tmr_Placing2
        OnMouseClick: write the text variable via Default
    Label (231,205 102x35), "Check Placing 3"
    RoundedRectangle (333,206 170x29), "%i ms", text variable: HMI_GVL.Tmr_Placing3
        OnMouseClick: write the text variable via Default
    Label (231,239 100x35), "Check Placing 4"
    RoundedRectangle (333,240 170x29), "%i ms", text variable: HMI_GVL.Tmr_Placing4
        OnMouseClick: write the text variable via Default
    Button (772,231 170x40), "Bypass FGHS", colour toggle: HMI_GVL.BypassFGHS, image: VisuSymbols.Symbols.Lock
        toggle HMI_GVL.BypassFGHS
END_VISUALIZATION

// ---- VISUs/Parameter/Recipe/MOffset_2.TcVIS
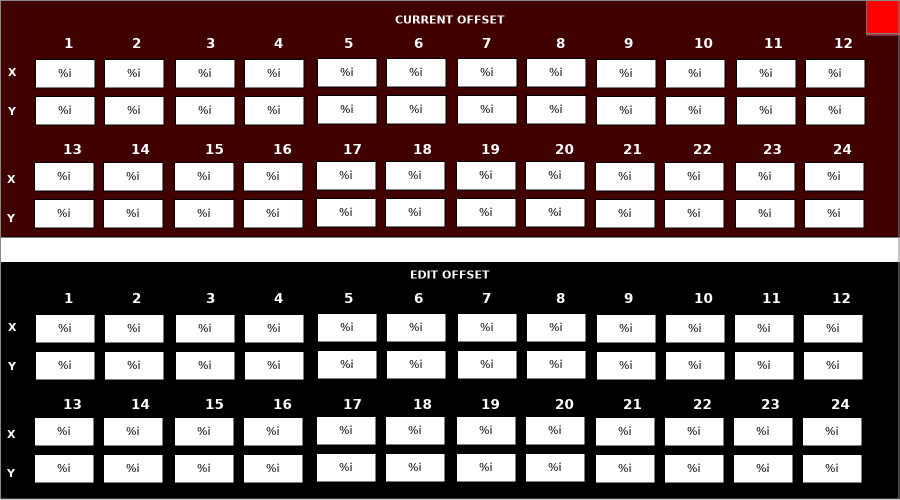
VISUALIZATION MOffset_2  // 900x500
    RoundedRectangle (0,0 900x237)
    Label (0,0 900x40), "CURRENT OFFSET"
    Label (5,55 25x35), "X"
    RoundedRectangle (35,59 60x29), "%i", text variable: Status_GVL.RecipeLine[2].OffsetPattern.Offset_X[1]
    Label (61,26 25x35), "1"
    RoundedRectangle (104,59 60x29), "%i", text variable: Status_GVL.RecipeLine[2].OffsetPattern.Offset_X[2]
    Label (129,26 25x35), "2"
    RoundedRectangle (175,59 60x29), "%i", text variable: Status_GVL.RecipeLine[2].OffsetPattern.Offset_X[3]
    RoundedRectangle (244,59 60x29), "%i", text variable: Status_GVL.RecipeLine[2].OffsetPattern.Offset_X[4]
    Label (5,94 25x35), "Y"
    RoundedRectangle (317,58 60x29), "%i", text variable: Status_GVL.RecipeLine[2].OffsetPattern.Offset_X[5]
    RoundedRectangle (386,58 60x29), "%i", text variable: Status_GVL.RecipeLine[2].OffsetPattern.Offset_X[6]
    RoundedRectangle (457,58 60x29), "%i", text variable: Status_GVL.RecipeLine[2].OffsetPattern.Offset_X[7]
    RoundedRectangle (526,58 60x29), "%i", text variable: Status_GVL.RecipeLine[2].OffsetPattern.Offset_X[8]
    RoundedRectangle (596,59 60x29), "%i", text variable: Status_GVL.RecipeLine[2].OffsetPattern.Offset_X[9]
    RoundedRectangle (665,59 60x29), "%i", text variable: Status_GVL.RecipeLine[2].OffsetPattern.Offset_X[10]
    Label (203,26 25x35), "3"
    Label (271,26 25x35), "4"
    Label (341,26 25x35), "5"
    Label (411,26 25x35), "6"
    Label (479,26 25x35), "7"
    Label (553,26 25x35), "8"
    Label (621,26 25x35), "9"
    Label (691,26 25x35), "10"
    RoundedRectangle (35,96 60x29), "%i", text variable: Status_GVL.RecipeLine[2].OffsetPattern.Offset_Y[1]
    RoundedRectangle (104,96 60x29), "%i", text variable: Status_GVL.RecipeLine[2].OffsetPattern.Offset_Y[2]
    RoundedRectangle (175,96 60x29), "%i", text variable: Status_GVL.RecipeLine[2].OffsetPattern.Offset_Y[3]
    RoundedRectangle (244,96 60x29), "%i", text variable: Status_GVL.RecipeLine[2].OffsetPattern.Offset_Y[4]
    RoundedRectangle (317,95 60x29), "%i", text variable: Status_GVL.RecipeLine[2].OffsetPattern.Offset_Y[5]
    RoundedRectangle (386,95 60x29), "%i", text variable: Status_GVL.RecipeLine[2].OffsetPattern.Offset_Y[6]
    RoundedRectangle (457,95 60x29), "%i", text variable: Status_GVL.RecipeLine[2].OffsetPattern.Offset_Y[7]
    RoundedRectangle (526,95 60x29), "%i", text variable: Status_GVL.RecipeLine[2].OffsetPattern.Offset_Y[8]
    RoundedRectangle (596,96 60x29), "%i", text variable: Status_GVL.RecipeLine[2].OffsetPattern.Offset_Y[9]
    RoundedRectangle (665,96 60x29), "%i", text variable: Status_GVL.RecipeLine[2].OffsetPattern.Offset_Y[10]
    Label (4,162 25x35), "X"
    RoundedRectangle (34,162 60x29), "%i", text variable: Status_GVL.RecipeLine[2].OffsetPattern.Offset_X[13]
    RoundedRectangle (103,162 60x29), "%i", text variable: Status_GVL.RecipeLine[2].OffsetPattern.Offset_X[14]
    RoundedRectangle (174,162 60x29), "%i", text variable: Status_GVL.RecipeLine[2].OffsetPattern.Offset_X[15]
    RoundedRectangle (243,162 60x29), "%i", text variable: Status_GVL.RecipeLine[2].OffsetPattern.Offset_X[16]
    Label (4,201 25x35), "Y"
    RoundedRectangle (316,161 60x29), "%i", text variable: Status_GVL.RecipeLine[2].OffsetPattern.Offset_X[17]
    RoundedRectangle (385,161 60x29), "%i", text variable: Status_GVL.RecipeLine[2].OffsetPattern.Offset_X[18]
    RoundedRectangle (456,161 60x29), "%i", text variable: Status_GVL.RecipeLine[2].OffsetPattern.Offset_X[19]
    RoundedRectangle (525,161 60x29), "%i", text variable: Status_GVL.RecipeLine[2].OffsetPattern.Offset_X[20]
    RoundedRectangle (595,162 60x29), "%i", text variable: Status_GVL.RecipeLine[2].OffsetPattern.Offset_X[21]
    RoundedRectangle (664,162 60x29), "%i", text variable: Status_GVL.RecipeLine[2].OffsetPattern.Offset_X[22]
    RoundedRectangle (34,199 60x29), "%i", text variable: Status_GVL.RecipeLine[2].OffsetPattern.Offset_Y[13]
    RoundedRectangle (103,199 60x29), "%i", text variable: Status_GVL.RecipeLine[2].OffsetPattern.Offset_Y[14]
    RoundedRectangle (174,199 60x29), "%i", text variable: Status_GVL.RecipeLine[2].OffsetPattern.Offset_Y[15]
    RoundedRectangle (243,199 60x29), "%i", text variable: Status_GVL.RecipeLine[2].OffsetPattern.Offset_Y[16]
    RoundedRectangle (316,198 60x29), "%i", text variable: Status_GVL.RecipeLine[2].OffsetPattern.Offset_Y[17]
    RoundedRectangle (385,198 60x29), "%i", text variable: Status_GVL.RecipeLine[2].OffsetPattern.Offset_Y[18]
    RoundedRectangle (456,198 60x29), "%i", text variable: Status_GVL.RecipeLine[2].OffsetPattern.Offset_Y[19]
    RoundedRectangle (525,198 60x29), "%i", text variable: Status_GVL.RecipeLine[2].OffsetPattern.Offset_Y[20]
    RoundedRectangle (595,199 60x29), "%i", text variable: Status_GVL.RecipeLine[2].OffsetPattern.Offset_Y[21]
    RoundedRectangle (664,199 60x29), "%i", text variable: Status_GVL.RecipeLine[2].OffsetPattern.Offset_Y[22]
    Label (60,132 25x35), "13"
    Label (128,132 25x35), "14"
    Label (202,132 25x35), "15"
    Label (270,132 25x35), "16"
    Label (340,132 25x35), "17"
    Label (410,132 25x35), "18"
    Label (478,132 25x35), "19"
    Label (552,132 25x35), "20"
    Label (620,132 25x35), "21"
    Label (690,132 25x35), "22"
    RoundedRectangle (0,262 900x237)
    Label (0,255 900x40), "EDIT OFFSET"
    Label (5,310 25x35), "X"
    RoundedRectangle (35,314 60x29), "%i", text variable: HMI_GVL.arRecipeHMI[2].OffsetPattern.Offset_X[1], input disabled if: Status_GVL.StsEdit[2]
        OnMouseClick: write the text variable via Default
    Label (61,281 25x35), "1"
    RoundedRectangle (104,314 60x29), "%i", text variable: HMI_GVL.arRecipeHMI[2].OffsetPattern.Offset_X[2], input disabled if: Status_GVL.StsEdit[2]
        OnMouseClick: write the text variable via Default
    Label (129,281 25x35), "2"
    RoundedRectangle (175,314 60x29), "%i", text variable: HMI_GVL.arRecipeHMI[2].OffsetPattern.Offset_X[3], input disabled if: Status_GVL.StsEdit[2]
        OnMouseClick: write the text variable via Default
    RoundedRectangle (244,314 60x29), "%i", text variable: HMI_GVL.arRecipeHMI[2].OffsetPattern.Offset_X[4], input disabled if: Status_GVL.StsEdit[2]
        OnMouseClick: write the text variable via Default
    Label (5,349 25x35), "Y"
    RoundedRectangle (317,313 60x29), "%i", text variable: HMI_GVL.arRecipeHMI[2].OffsetPattern.Offset_X[5], input disabled if: Status_GVL.StsEdit[2]
        OnMouseClick: write the text variable via Default
    RoundedRectangle (386,313 60x29), "%i", text variable: HMI_GVL.arRecipeHMI[2].OffsetPattern.Offset_X[6], input disabled if: Status_GVL.StsEdit[2]
        OnMouseClick: write the text variable via Default
    RoundedRectangle (457,313 60x29), "%i", text variable: HMI_GVL.arRecipeHMI[2].OffsetPattern.Offset_X[7], input disabled if: Status_GVL.StsEdit[2]
        OnMouseClick: write the text variable via Default
    RoundedRectangle (526,313 60x29), "%i", text variable: HMI_GVL.arRecipeHMI[2].OffsetPattern.Offset_X[8], input disabled if: Status_GVL.StsEdit[2]
        OnMouseClick: write the text variable via Default
    RoundedRectangle (596,314 60x29), "%i", text variable: HMI_GVL.arRecipeHMI[2].OffsetPattern.Offset_X[9], input disabled if: Status_GVL.StsEdit[2]
        OnMouseClick: write the text variable via Default
    RoundedRectangle (665,314 60x29), "%i", text variable: HMI_GVL.arRecipeHMI[2].OffsetPattern.Offset_X[10], input disabled if: Status_GVL.StsEdit[2]
        OnMouseClick: write the text variable via Default
    Label (203,281 25x35), "3"
    Label (271,281 25x35), "4"
    Label (341,281 25x35), "5"
    Label (411,281 25x35), "6"
    Label (479,281 25x35), "7"
    Label (553,281 25x35), "8"
    Label (621,281 25x35), "9"
    Label (691,281 25x35), "10"
    RoundedRectangle (35,351 60x29), "%i", text variable: HMI_GVL.arRecipeHMI[2].OffsetPattern.Offset_Y[1], input disabled if: Status_GVL.StsEdit[2]
        OnMouseClick: write the text variable via Default
    RoundedRectangle (104,351 60x29), "%i", text variable: HMI_GVL.arRecipeHMI[2].OffsetPattern.Offset_Y[2], input disabled if: Status_GVL.StsEdit[2]
        OnMouseClick: write the text variable via Default
    RoundedRectangle (175,351 60x29), "%i", text variable: HMI_GVL.arRecipeHMI[2].OffsetPattern.Offset_Y[3], input disabled if: Status_GVL.StsEdit[2]
        OnMouseClick: write the text variable via Default
    RoundedRectangle (244,351 60x29), "%i", text variable: HMI_GVL.arRecipeHMI[2].OffsetPattern.Offset_Y[4], input disabled if: Status_GVL.StsEdit[2]
        OnMouseClick: write the text variable via Default
    RoundedRectangle (317,350 60x29), "%i", text variable: HMI_GVL.arRecipeHMI[2].OffsetPattern.Offset_Y[5], input disabled if: Status_GVL.StsEdit[2]
        OnMouseClick: write the text variable via Default
    RoundedRectangle (386,350 60x29), "%i", text variable: HMI_GVL.arRecipeHMI[2].OffsetPattern.Offset_Y[6], input disabled if: Status_GVL.StsEdit[2]
        OnMouseClick: write the text variable via Default
    RoundedRectangle (457,350 60x29), "%i", text variable: HMI_GVL.arRecipeHMI[2].OffsetPattern.Offset_Y[7], input disabled if: Status_GVL.StsEdit[2]
        OnMouseClick: write the text variable via Default
    RoundedRectangle (526,350 60x29), "%i", text variable: HMI_GVL.arRecipeHMI[2].OffsetPattern.Offset_Y[8], input disabled if: Status_GVL.StsEdit[2]
        OnMouseClick: write the text variable via Default
    RoundedRectangle (596,351 60x29), "%i", text variable: HMI_GVL.arRecipeHMI[2].OffsetPattern.Offset_Y[9], input disabled if: Status_GVL.StsEdit[2]
        OnMouseClick: write the text variable via Default
    RoundedRectangle (665,351 60x29), "%i", text variable: HMI_GVL.arRecipeHMI[2].OffsetPattern.Offset_Y[10], input disabled if: Status_GVL.StsEdit[2]
        OnMouseClick: write the text variable via Default
    Label (4,417 25x35), "X"
    RoundedRectangle (34,417 60x29), "%i", text variable: HMI_GVL.arRecipeHMI[2].OffsetPattern.Offset_X[13], input disabled if: Status_GVL.StsEdit[2]
        OnMouseClick: write the text variable via Default
    RoundedRectangle (103,417 60x29), "%i", text variable: HMI_GVL.arRecipeHMI[2].OffsetPattern.Offset_X[14], input disabled if: Status_GVL.StsEdit[2]
        OnMouseClick: write the text variable via Default
    RoundedRectangle (174,417 60x29), "%i", text variable: HMI_GVL.arRecipeHMI[2].OffsetPattern.Offset_X[15], input disabled if: Status_GVL.StsEdit[2]
        OnMouseClick: write the text variable via Default
    RoundedRectangle (243,417 60x29), "%i", text variable: HMI_GVL.arRecipeHMI[2].OffsetPattern.Offset_X[16], input disabled if: Status_GVL.StsEdit[2]
        OnMouseClick: write the text variable via Default
    Label (4,456 25x35), "Y"
    RoundedRectangle (316,416 60x29), "%i", text variable: HMI_GVL.arRecipeHMI[2].OffsetPattern.Offset_X[17], input disabled if: Status_GVL.StsEdit[2]
        OnMouseClick: write the text variable via Default
    RoundedRectangle (385,416 60x29), "%i", text variable: HMI_GVL.arRecipeHMI[2].OffsetPattern.Offset_X[18], input disabled if: Status_GVL.StsEdit[2]
        OnMouseClick: write the text variable via Default
    RoundedRectangle (456,416 60x29), "%i", text variable: HMI_GVL.arRecipeHMI[2].OffsetPattern.Offset_X[19], input disabled if: Status_GVL.StsEdit[2]
        OnMouseClick: write the text variable via Default
    RoundedRectangle (525,416 60x29), "%i", text variable: HMI_GVL.arRecipeHMI[2].OffsetPattern.Offset_X[20], input disabled if: Status_GVL.StsEdit[2]
        OnMouseClick: write the text variable via Default
    RoundedRectangle (595,417 60x29), "%i", text variable: HMI_GVL.arRecipeHMI[2].OffsetPattern.Offset_X[21], input disabled if: Status_GVL.StsEdit[2]
        OnMouseClick: write the text variable via Default
    RoundedRectangle (664,417 60x29), "%i", text variable: HMI_GVL.arRecipeHMI[2].OffsetPattern.Offset_X[22], input disabled if: Status_GVL.StsEdit[2]
        OnMouseClick: write the text variable via Default
    RoundedRectangle (34,454 60x29), "%i", text variable: HMI_GVL.arRecipeHMI[2].OffsetPattern.Offset_Y[13], input disabled if: Status_GVL.StsEdit[2]
        OnMouseClick: write the text variable via Default
    RoundedRectangle (103,454 60x29), "%i", text variable: HMI_GVL.arRecipeHMI[2].OffsetPattern.Offset_Y[14], input disabled if: Status_GVL.StsEdit[2]
        OnMouseClick: write the text variable via Default
    RoundedRectangle (174,454 60x29), "%i", text variable: HMI_GVL.arRecipeHMI[2].OffsetPattern.Offset_Y[15], input disabled if: Status_GVL.StsEdit[2]
        OnMouseClick: write the text variable via Default
    RoundedRectangle (243,454 60x29), "%i", text variable: HMI_GVL.arRecipeHMI[2].OffsetPattern.Offset_Y[16], input disabled if: Status_GVL.StsEdit[2]
        OnMouseClick: write the text variable via Default
    RoundedRectangle (316,453 60x29), "%i", text variable: HMI_GVL.arRecipeHMI[2].OffsetPattern.Offset_Y[17], input disabled if: Status_GVL.StsEdit[2]
        OnMouseClick: write the text variable via Default
    RoundedRectangle (385,453 60x29), "%i", text variable: HMI_GVL.arRecipeHMI[2].OffsetPattern.Offset_Y[18], input disabled if: Status_GVL.StsEdit[2]
        OnMouseClick: write the text variable via Default
    RoundedRectangle (456,453 60x29), "%i", text variable: HMI_GVL.arRecipeHMI[2].OffsetPattern.Offset_Y[19], input disabled if: Status_GVL.StsEdit[2]
        OnMouseClick: write the text variable via Default
    RoundedRectangle (525,453 60x29), "%i", text variable: HMI_GVL.arRecipeHMI[2].OffsetPattern.Offset_Y[20], input disabled if: Status_GVL.StsEdit[2]
        OnMouseClick: write the text variable via Default
    RoundedRectangle (595,454 60x29), "%i", text variable: HMI_GVL.arRecipeHMI[2].OffsetPattern.Offset_Y[21], input disabled if: Status_GVL.StsEdit[2]
        OnMouseClick: write the text variable via Default
    RoundedRectangle (664,454 60x29), "%i", text variable: HMI_GVL.arRecipeHMI[2].OffsetPattern.Offset_Y[22], input disabled if: Status_GVL.StsEdit[2]
        OnMouseClick: write the text variable via Default
    Label (60,387 25x35), "13"
    Label (128,387 25x35), "14"
    Label (202,387 25x35), "15"
    Label (270,387 25x35), "16"
    Label (340,387 25x35), "17"
    Label (410,387 25x35), "18"
    Label (478,387 25x35), "19"
    Label (552,387 25x35), "20"
    Label (620,387 25x35), "21"
    Label (690,387 25x35), "22"
    Button (866,0 35x35), image: VisuSymbols.Symbols.Wrong
        OnMouseClick: CloseDialog Dialog=MOffset_2, Result=OK, NumpadKeypadSet=True
    RoundedRectangle (736,59 60x29), "%i", text variable: Status_GVL.RecipeLine[2].OffsetPattern.Offset_X[11]
    RoundedRectangle (805,59 60x29), "%i", text variable: Status_GVL.RecipeLine[2].OffsetPattern.Offset_X[12]
    Label (761,26 25x35), "11"
    Label (831,26 25x35), "12"
    RoundedRectangle (736,96 60x29), "%i", text variable: Status_GVL.RecipeLine[2].OffsetPattern.Offset_Y[11]
    RoundedRectangle (805,96 60x29), "%i", text variable: Status_GVL.RecipeLine[2].OffsetPattern.Offset_Y[12]
    RoundedRectangle (735,162 60x29), "%i", text variable: Status_GVL.RecipeLine[2].OffsetPattern.Offset_X[23]
    RoundedRectangle (804,162 60x29), "%i", text variable: Status_GVL.RecipeLine[2].OffsetPattern.Offset_X[24]
    RoundedRectangle (735,199 60x29), "%i", text variable: Status_GVL.RecipeLine[2].OffsetPattern.Offset_Y[23]
    RoundedRectangle (804,199 60x29), "%i", text variable: Status_GVL.RecipeLine[2].OffsetPattern.Offset_Y[24]
    Label (760,132 25x35), "23"
    Label (830,132 25x35), "24"
    RoundedRectangle (734,314 60x29), "%i", text variable: HMI_GVL.arRecipeHMI[2].OffsetPattern.Offset_X[11], input disabled if: Status_GVL.StsEdit[2]
        OnMouseClick: write the text variable via Default
    RoundedRectangle (803,314 60x29), "%i", text variable: HMI_GVL.arRecipeHMI[2].OffsetPattern.Offset_X[12], input disabled if: Status_GVL.StsEdit[2]
        OnMouseClick: write the text variable via Default
    Label (759,281 25x35), "11"
    Label (829,281 25x35), "12"
    RoundedRectangle (734,351 60x29), "%i", text variable: HMI_GVL.arRecipeHMI[2].OffsetPattern.Offset_Y[11], input disabled if: Status_GVL.StsEdit[2]
        OnMouseClick: write the text variable via Default
    RoundedRectangle (803,351 60x29), "%i", text variable: HMI_GVL.arRecipeHMI[2].OffsetPattern.Offset_Y[12], input disabled if: Status_GVL.StsEdit[2]
        OnMouseClick: write the text variable via Default
    RoundedRectangle (733,417 60x29), "%i", text variable: HMI_GVL.arRecipeHMI[2].OffsetPattern.Offset_X[23], input disabled if: Status_GVL.StsEdit[2]
        OnMouseClick: write the text variable via Default
    RoundedRectangle (802,417 60x29), "%i", text variable: HMI_GVL.arRecipeHMI[2].OffsetPattern.Offset_X[24], input disabled if: Status_GVL.StsEdit[2]
        OnMouseClick: write the text variable via Default
    RoundedRectangle (733,454 60x29), "%i", text variable: HMI_GVL.arRecipeHMI[2].OffsetPattern.Offset_Y[23], input disabled if: Status_GVL.StsEdit[2]
        OnMouseClick: write the text variable via Default
    RoundedRectangle (802,454 60x29), "%i", text variable: HMI_GVL.arRecipeHMI[2].OffsetPattern.Offset_Y[24], input disabled if: Status_GVL.StsEdit[2]
        OnMouseClick: write the text variable via Default
    Label (758,387 25x35), "23"
    Label (828,387 25x35), "24"
END_VISUALIZATION

// ---- VISUs/Parameter/Recipe/MOffset_3.TcVIS
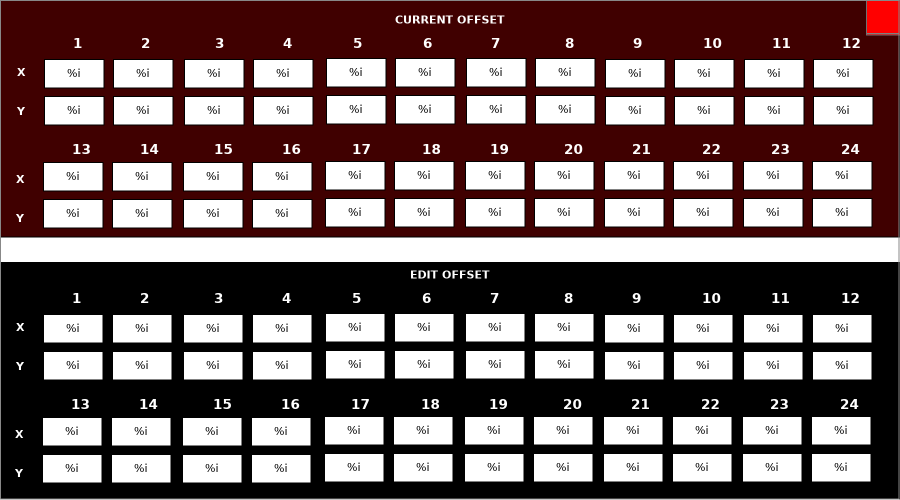
VISUALIZATION MOffset_3  // 900x500
    RoundedRectangle (0,0 900x237)
    Label (0,0 900x40), "CURRENT OFFSET"
    Label (14,55 25x35), "X"
    RoundedRectangle (44,59 60x29), "%i", text variable: Status_GVL.RecipeLine[3].OffsetPattern.Offset_X[1]
    Label (70,26 25x35), "1"
    RoundedRectangle (113,59 60x29), "%i", text variable: Status_GVL.RecipeLine[3].OffsetPattern.Offset_X[2]
    Label (138,26 25x35), "2"
    RoundedRectangle (184,59 60x29), "%i", text variable: Status_GVL.RecipeLine[3].OffsetPattern.Offset_X[3]
    RoundedRectangle (253,59 60x29), "%i", text variable: Status_GVL.RecipeLine[3].OffsetPattern.Offset_X[4]
    Label (14,94 25x35), "Y"
    RoundedRectangle (326,58 60x29), "%i", text variable: Status_GVL.RecipeLine[3].OffsetPattern.Offset_X[5]
    RoundedRectangle (395,58 60x29), "%i", text variable: Status_GVL.RecipeLine[3].OffsetPattern.Offset_X[6]
    RoundedRectangle (466,58 60x29), "%i", text variable: Status_GVL.RecipeLine[3].OffsetPattern.Offset_X[7]
    RoundedRectangle (535,58 60x29), "%i", text variable: Status_GVL.RecipeLine[3].OffsetPattern.Offset_X[8]
    RoundedRectangle (605,59 60x29), "%i", text variable: Status_GVL.RecipeLine[3].OffsetPattern.Offset_X[9]
    RoundedRectangle (674,59 60x29), "%i", text variable: Status_GVL.RecipeLine[3].OffsetPattern.Offset_X[10]
    Label (212,26 25x35), "3"
    Label (280,26 25x35), "4"
    Label (350,26 25x35), "5"
    Label (420,26 25x35), "6"
    Label (488,26 25x35), "7"
    Label (562,26 25x35), "8"
    Label (630,26 25x35), "9"
    Label (700,26 25x35), "10"
    RoundedRectangle (44,96 60x29), "%i", text variable: Status_GVL.RecipeLine[3].OffsetPattern.Offset_Y[1]
    RoundedRectangle (113,96 60x29), "%i", text variable: Status_GVL.RecipeLine[3].OffsetPattern.Offset_Y[2]
    RoundedRectangle (184,96 60x29), "%i", text variable: Status_GVL.RecipeLine[3].OffsetPattern.Offset_Y[3]
    RoundedRectangle (253,96 60x29), "%i", text variable: Status_GVL.RecipeLine[3].OffsetPattern.Offset_Y[4]
    RoundedRectangle (326,95 60x29), "%i", text variable: Status_GVL.RecipeLine[3].OffsetPattern.Offset_Y[5]
    RoundedRectangle (395,95 60x29), "%i", text variable: Status_GVL.RecipeLine[3].OffsetPattern.Offset_Y[6]
    RoundedRectangle (466,95 60x29), "%i", text variable: Status_GVL.RecipeLine[3].OffsetPattern.Offset_Y[7]
    RoundedRectangle (535,95 60x29), "%i", text variable: Status_GVL.RecipeLine[3].OffsetPattern.Offset_Y[8]
    RoundedRectangle (605,96 60x29), "%i", text variable: Status_GVL.RecipeLine[3].OffsetPattern.Offset_Y[9]
    RoundedRectangle (674,96 60x29), "%i", text variable: Status_GVL.RecipeLine[3].OffsetPattern.Offset_Y[10]
    Label (13,162 25x35), "X"
    RoundedRectangle (43,162 60x29), "%i", text variable: Status_GVL.RecipeLine[3].OffsetPattern.Offset_X[13]
    RoundedRectangle (112,162 60x29), "%i", text variable: Status_GVL.RecipeLine[3].OffsetPattern.Offset_X[14]
    RoundedRectangle (183,162 60x29), "%i", text variable: Status_GVL.RecipeLine[3].OffsetPattern.Offset_X[15]
    RoundedRectangle (252,162 60x29), "%i", text variable: Status_GVL.RecipeLine[3].OffsetPattern.Offset_X[16]
    Label (13,201 25x35), "Y"
    RoundedRectangle (325,161 60x29), "%i", text variable: Status_GVL.RecipeLine[3].OffsetPattern.Offset_X[17]
    RoundedRectangle (394,161 60x29), "%i", text variable: Status_GVL.RecipeLine[3].OffsetPattern.Offset_X[18]
    RoundedRectangle (465,161 60x29), "%i", text variable: Status_GVL.RecipeLine[3].OffsetPattern.Offset_X[19]
    RoundedRectangle (534,161 60x29), "%i", text variable: Status_GVL.RecipeLine[3].OffsetPattern.Offset_X[20]
    RoundedRectangle (604,161 60x29), "%i", text variable: Status_GVL.RecipeLine[3].OffsetPattern.Offset_X[21]
    RoundedRectangle (673,161 60x29), "%i", text variable: Status_GVL.RecipeLine[3].OffsetPattern.Offset_X[22]
    RoundedRectangle (43,199 60x29), "%i", text variable: Status_GVL.RecipeLine[3].OffsetPattern.Offset_Y[13]
    RoundedRectangle (112,199 60x29), "%i", text variable: Status_GVL.RecipeLine[3].OffsetPattern.Offset_Y[14]
    RoundedRectangle (183,199 60x29), "%i", text variable: Status_GVL.RecipeLine[3].OffsetPattern.Offset_Y[15]
    RoundedRectangle (252,199 60x29), "%i", text variable: Status_GVL.RecipeLine[3].OffsetPattern.Offset_Y[16]
    RoundedRectangle (325,198 60x29), "%i", text variable: Status_GVL.RecipeLine[3].OffsetPattern.Offset_Y[17]
    RoundedRectangle (394,198 60x29), "%i", text variable: Status_GVL.RecipeLine[3].OffsetPattern.Offset_Y[18]
    RoundedRectangle (465,198 60x29), "%i", text variable: Status_GVL.RecipeLine[3].OffsetPattern.Offset_Y[19]
    RoundedRectangle (534,198 60x29), "%i", text variable: Status_GVL.RecipeLine[3].OffsetPattern.Offset_Y[20]
    RoundedRectangle (604,198 60x29), "%i", text variable: Status_GVL.RecipeLine[3].OffsetPattern.Offset_Y[21]
    RoundedRectangle (673,198 60x29), "%i", text variable: Status_GVL.RecipeLine[3].OffsetPattern.Offset_Y[22]
    Label (69,132 25x35), "13"
    Label (137,132 25x35), "14"
    Label (211,132 25x35), "15"
    Label (279,132 25x35), "16"
    Label (349,132 25x35), "17"
    Label (419,132 25x35), "18"
    Label (487,132 25x35), "19"
    Label (561,132 25x35), "20"
    Label (629,132 25x35), "21"
    Label (699,132 25x35), "22"
    RoundedRectangle (0,262 900x237)
    Label (0,255 900x40), "EDIT OFFSET"
    Label (13,310 25x35), "X"
    RoundedRectangle (43,314 60x29), "%i", text variable: HMI_GVL.arRecipeHMI[3].OffsetPattern.Offset_X[1], input disabled if: Status_GVL.StsEdit[3]
        OnMouseClick: write the text variable via Default
    Label (69,281 25x35), "1"
    RoundedRectangle (112,314 60x29), "%i", text variable: HMI_GVL.arRecipeHMI[3].OffsetPattern.Offset_X[2], input disabled if: Status_GVL.StsEdit[3]
        OnMouseClick: write the text variable via Default
    Label (137,281 25x35), "2"
    RoundedRectangle (183,314 60x29), "%i", text variable: HMI_GVL.arRecipeHMI[3].OffsetPattern.Offset_X[3], input disabled if: Status_GVL.StsEdit[3]
        OnMouseClick: write the text variable via Default
    RoundedRectangle (252,314 60x29), "%i", text variable: HMI_GVL.arRecipeHMI[3].OffsetPattern.Offset_X[4], input disabled if: Status_GVL.StsEdit[3]
        OnMouseClick: write the text variable via Default
    Label (13,349 25x35), "Y"
    RoundedRectangle (325,313 60x29), "%i", text variable: HMI_GVL.arRecipeHMI[3].OffsetPattern.Offset_X[5], input disabled if: Status_GVL.StsEdit[3]
        OnMouseClick: write the text variable via Default
    RoundedRectangle (394,313 60x29), "%i", text variable: HMI_GVL.arRecipeHMI[3].OffsetPattern.Offset_X[6], input disabled if: Status_GVL.StsEdit[3]
        OnMouseClick: write the text variable via Default
    RoundedRectangle (465,313 60x29), "%i", text variable: HMI_GVL.arRecipeHMI[3].OffsetPattern.Offset_X[7], input disabled if: Status_GVL.StsEdit[3]
        OnMouseClick: write the text variable via Default
    RoundedRectangle (534,313 60x29), "%i", text variable: HMI_GVL.arRecipeHMI[3].OffsetPattern.Offset_X[8], input disabled if: Status_GVL.StsEdit[3]
        OnMouseClick: write the text variable via Default
    RoundedRectangle (604,314 60x29), "%i", text variable: HMI_GVL.arRecipeHMI[3].OffsetPattern.Offset_X[9], input disabled if: Status_GVL.StsEdit[3]
        OnMouseClick: write the text variable via Default
    RoundedRectangle (673,314 60x29), "%i", text variable: HMI_GVL.arRecipeHMI[3].OffsetPattern.Offset_X[10], input disabled if: Status_GVL.StsEdit[3]
        OnMouseClick: write the text variable via Default
    Label (211,281 25x35), "3"
    Label (279,281 25x35), "4"
    Label (349,281 25x35), "5"
    Label (419,281 25x35), "6"
    Label (487,281 25x35), "7"
    Label (561,281 25x35), "8"
    Label (629,281 25x35), "9"
    Label (699,281 25x35), "10"
    RoundedRectangle (43,351 60x29), "%i", text variable: HMI_GVL.arRecipeHMI[3].OffsetPattern.Offset_Y[1], input disabled if: Status_GVL.StsEdit[3]
        OnMouseClick: write the text variable via Default
    RoundedRectangle (112,351 60x29), "%i", text variable: HMI_GVL.arRecipeHMI[3].OffsetPattern.Offset_Y[2], input disabled if: Status_GVL.StsEdit[3]
        OnMouseClick: write the text variable via Default
    RoundedRectangle (183,351 60x29), "%i", text variable: HMI_GVL.arRecipeHMI[3].OffsetPattern.Offset_Y[3], input disabled if: Status_GVL.StsEdit[3]
        OnMouseClick: write the text variable via Default
    RoundedRectangle (252,351 60x29), "%i", text variable: HMI_GVL.arRecipeHMI[3].OffsetPattern.Offset_Y[4], input disabled if: Status_GVL.StsEdit[3]
        OnMouseClick: write the text variable via Default
    RoundedRectangle (325,350 60x29), "%i", text variable: HMI_GVL.arRecipeHMI[3].OffsetPattern.Offset_Y[5], input disabled if: Status_GVL.StsEdit[3]
        OnMouseClick: write the text variable via Default
    RoundedRectangle (394,350 60x29), "%i", text variable: HMI_GVL.arRecipeHMI[3].OffsetPattern.Offset_Y[6], input disabled if: Status_GVL.StsEdit[3]
        OnMouseClick: write the text variable via Default
    RoundedRectangle (465,350 60x29), "%i", text variable: HMI_GVL.arRecipeHMI[3].OffsetPattern.Offset_Y[7], input disabled if: Status_GVL.StsEdit[3]
        OnMouseClick: write the text variable via Default
    RoundedRectangle (534,350 60x29), "%i", text variable: HMI_GVL.arRecipeHMI[3].OffsetPattern.Offset_Y[8], input disabled if: Status_GVL.StsEdit[3]
        OnMouseClick: write the text variable via Default
    RoundedRectangle (604,351 60x29), "%i", text variable: HMI_GVL.arRecipeHMI[3].OffsetPattern.Offset_Y[9], input disabled if: Status_GVL.StsEdit[3]
        OnMouseClick: write the text variable via Default
    RoundedRectangle (673,351 60x29), "%i", text variable: HMI_GVL.arRecipeHMI[3].OffsetPattern.Offset_Y[10], input disabled if: Status_GVL.StsEdit[3]
        OnMouseClick: write the text variable via Default
    Label (12,417 25x35), "X"
    RoundedRectangle (42,417 60x29), "%i", text variable: HMI_GVL.arRecipeHMI[3].OffsetPattern.Offset_X[13], input disabled if: Status_GVL.StsEdit[3]
        OnMouseClick: write the text variable via Default
    RoundedRectangle (111,417 60x29), "%i", text variable: HMI_GVL.arRecipeHMI[3].OffsetPattern.Offset_X[14], input disabled if: Status_GVL.StsEdit[3]
        OnMouseClick: write the text variable via Default
    RoundedRectangle (182,417 60x29), "%i", text variable: HMI_GVL.arRecipeHMI[3].OffsetPattern.Offset_X[15], input disabled if: Status_GVL.StsEdit[3]
        OnMouseClick: write the text variable via Default
    RoundedRectangle (251,417 60x29), "%i", text variable: HMI_GVL.arRecipeHMI[3].OffsetPattern.Offset_X[16], input disabled if: Status_GVL.StsEdit[3]
        OnMouseClick: write the text variable via Default
    Label (12,456 25x35), "Y"
    RoundedRectangle (324,416 60x29), "%i", text variable: HMI_GVL.arRecipeHMI[3].OffsetPattern.Offset_X[17], input disabled if: Status_GVL.StsEdit[3]
        OnMouseClick: write the text variable via Default
    RoundedRectangle (393,416 60x29), "%i", text variable: HMI_GVL.arRecipeHMI[3].OffsetPattern.Offset_X[18], input disabled if: Status_GVL.StsEdit[3]
        OnMouseClick: write the text variable via Default
    RoundedRectangle (464,416 60x29), "%i", text variable: HMI_GVL.arRecipeHMI[3].OffsetPattern.Offset_X[19], input disabled if: Status_GVL.StsEdit[3]
        OnMouseClick: write the text variable via Default
    RoundedRectangle (533,416 60x29), "%i", text variable: HMI_GVL.arRecipeHMI[3].OffsetPattern.Offset_X[20], input disabled if: Status_GVL.StsEdit[3]
        OnMouseClick: write the text variable via Default
    RoundedRectangle (603,416 60x29), "%i", text variable: HMI_GVL.arRecipeHMI[3].OffsetPattern.Offset_X[21], input disabled if: Status_GVL.StsEdit[3]
        OnMouseClick: write the text variable via Default
    RoundedRectangle (672,416 60x29), "%i", text variable: HMI_GVL.arRecipeHMI[3].OffsetPattern.Offset_X[22], input disabled if: Status_GVL.StsEdit[3]
        OnMouseClick: write the text variable via Default
    RoundedRectangle (42,454 60x29), "%i", text variable: HMI_GVL.arRecipeHMI[3].OffsetPattern.Offset_Y[13], input disabled if: Status_GVL.StsEdit[3]
        OnMouseClick: write the text variable via Default
    RoundedRectangle (111,454 60x29), "%i", text variable: HMI_GVL.arRecipeHMI[3].OffsetPattern.Offset_Y[14], input disabled if: Status_GVL.StsEdit[3]
        OnMouseClick: write the text variable via Default
    RoundedRectangle (182,454 60x29), "%i", text variable: HMI_GVL.arRecipeHMI[3].OffsetPattern.Offset_Y[15], input disabled if: Status_GVL.StsEdit[3]
        OnMouseClick: write the text variable via Default
    RoundedRectangle (251,454 60x29), "%i", text variable: HMI_GVL.arRecipeHMI[3].OffsetPattern.Offset_Y[16], input disabled if: Status_GVL.StsEdit[3]
        OnMouseClick: write the text variable via Default
    RoundedRectangle (324,453 60x29), "%i", text variable: HMI_GVL.arRecipeHMI[3].OffsetPattern.Offset_Y[17], input disabled if: Status_GVL.StsEdit[3]
        OnMouseClick: write the text variable via Default
    RoundedRectangle (393,453 60x29), "%i", text variable: HMI_GVL.arRecipeHMI[3].OffsetPattern.Offset_Y[18], input disabled if: Status_GVL.StsEdit[3]
        OnMouseClick: write the text variable via Default
    RoundedRectangle (464,453 60x29), "%i", text variable: HMI_GVL.arRecipeHMI[3].OffsetPattern.Offset_Y[19], input disabled if: Status_GVL.StsEdit[3]
        OnMouseClick: write the text variable via Default
    RoundedRectangle (533,453 60x29), "%i", text variable: HMI_GVL.arRecipeHMI[3].OffsetPattern.Offset_Y[20], input disabled if: Status_GVL.StsEdit[3]
        OnMouseClick: write the text variable via Default
    RoundedRectangle (603,453 60x29), "%i", text variable: HMI_GVL.arRecipeHMI[3].OffsetPattern.Offset_Y[21], input disabled if: Status_GVL.StsEdit[3]
        OnMouseClick: write the text variable via Default
    RoundedRectangle (672,453 60x29), "%i", text variable: HMI_GVL.arRecipeHMI[3].OffsetPattern.Offset_Y[22], input disabled if: Status_GVL.StsEdit[3]
        OnMouseClick: write the text variable via Default
    Label (68,387 25x35), "13"
    Label (136,387 25x35), "14"
    Label (210,387 25x35), "15"
    Label (278,387 25x35), "16"
    Label (348,387 25x35), "17"
    Label (418,387 25x35), "18"
    Label (486,387 25x35), "19"
    Label (560,387 25x35), "20"
    Label (628,387 25x35), "21"
    Label (698,387 25x35), "22"
    Button (866,0 35x35), image: VisuSymbols.Symbols.Wrong
        OnMouseClick: CloseDialog Dialog=MOffset_3, Result=OK, NumpadKeypadSet=True
    RoundedRectangle (744,59 60x29), "%i", text variable: Status_GVL.RecipeLine[3].OffsetPattern.Offset_X[11]
    RoundedRectangle (813,59 60x29), "%i", text variable: Status_GVL.RecipeLine[3].OffsetPattern.Offset_X[12]
    Label (769,26 25x35), "11"
    Label (839,26 25x35), "12"
    RoundedRectangle (744,96 60x29), "%i", text variable: Status_GVL.RecipeLine[3].OffsetPattern.Offset_Y[11]
    RoundedRectangle (813,96 60x29), "%i", text variable: Status_GVL.RecipeLine[3].OffsetPattern.Offset_Y[12]
    RoundedRectangle (743,161 60x29), "%i", text variable: Status_GVL.RecipeLine[3].OffsetPattern.Offset_X[23]
    RoundedRectangle (812,161 60x29), "%i", text variable: Status_GVL.RecipeLine[3].OffsetPattern.Offset_X[24]
    RoundedRectangle (743,198 60x29), "%i", text variable: Status_GVL.RecipeLine[3].OffsetPattern.Offset_Y[23]
    RoundedRectangle (812,198 60x29), "%i", text variable: Status_GVL.RecipeLine[3].OffsetPattern.Offset_Y[24]
    Label (768,132 25x35), "23"
    Label (838,132 25x35), "24"
    RoundedRectangle (743,314 60x29), "%i", text variable: HMI_GVL.arRecipeHMI[3].OffsetPattern.Offset_X[11], input disabled if: Status_GVL.StsEdit[3]
        OnMouseClick: write the text variable via Default
    RoundedRectangle (812,314 60x29), "%i", text variable: HMI_GVL.arRecipeHMI[3].OffsetPattern.Offset_X[12], input disabled if: Status_GVL.StsEdit[3]
        OnMouseClick: write the text variable via Default
    Label (768,281 25x35), "11"
    Label (838,281 25x35), "12"
    RoundedRectangle (743,351 60x29), "%i", text variable: HMI_GVL.arRecipeHMI[3].OffsetPattern.Offset_Y[11], input disabled if: Status_GVL.StsEdit[3]
        OnMouseClick: write the text variable via Default
    RoundedRectangle (812,351 60x29), "%i", text variable: HMI_GVL.arRecipeHMI[3].OffsetPattern.Offset_Y[12], input disabled if: Status_GVL.StsEdit[3]
        OnMouseClick: write the text variable via Default
    RoundedRectangle (742,416 60x29), "%i", text variable: HMI_GVL.arRecipeHMI[3].OffsetPattern.Offset_X[23], input disabled if: Status_GVL.StsEdit[3]
        OnMouseClick: write the text variable via Default
    RoundedRectangle (811,416 60x29), "%i", text variable: HMI_GVL.arRecipeHMI[3].OffsetPattern.Offset_X[24], input disabled if: Status_GVL.StsEdit[3]
        OnMouseClick: write the text variable via Default
    RoundedRectangle (742,453 60x29), "%i", text variable: HMI_GVL.arRecipeHMI[3].OffsetPattern.Offset_Y[23], input disabled if: Status_GVL.StsEdit[3]
        OnMouseClick: write the text variable via Default
    RoundedRectangle (811,453 60x29), "%i", text variable: HMI_GVL.arRecipeHMI[3].OffsetPattern.Offset_Y[24], input disabled if: Status_GVL.StsEdit[3]
        OnMouseClick: write the text variable via Default
    Label (767,387 25x35), "23"
    Label (837,387 25x35), "24"
END_VISUALIZATION

// ---- VISUs/Parameter/Recipe/MOffset_4.TcVIS
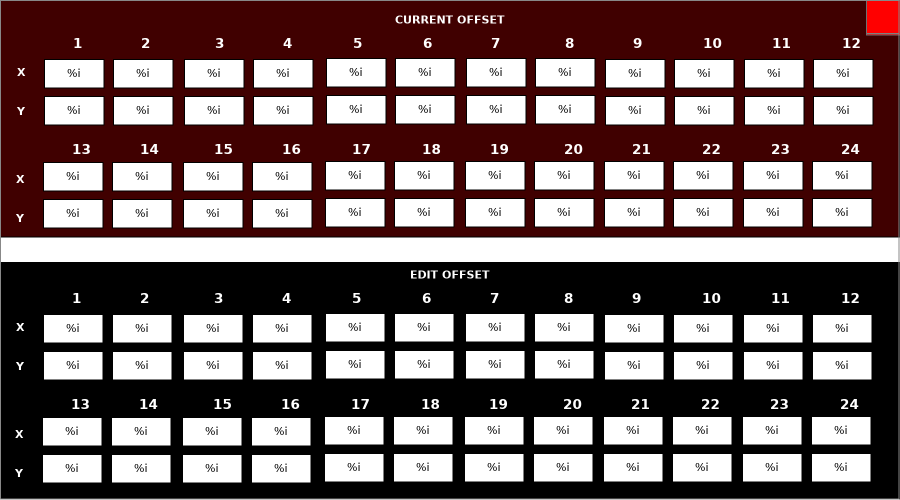
VISUALIZATION MOffset_4  // 900x500
    RoundedRectangle (0,0 900x237)
    Label (0,0 900x40), "CURRENT OFFSET"
    Label (14,55 25x35), "X"
    RoundedRectangle (44,59 60x29), "%i", text variable: Status_GVL.RecipeLine[4].OffsetPattern.Offset_X[1]
    Label (70,26 25x35), "1"
    RoundedRectangle (113,59 60x29), "%i", text variable: Status_GVL.RecipeLine[4].OffsetPattern.Offset_X[2]
    Label (138,26 25x35), "2"
    RoundedRectangle (184,59 60x29), "%i", text variable: Status_GVL.RecipeLine[4].OffsetPattern.Offset_X[3]
    RoundedRectangle (253,59 60x29), "%i", text variable: Status_GVL.RecipeLine[4].OffsetPattern.Offset_X[4]
    Label (14,94 25x35), "Y"
    RoundedRectangle (326,58 60x29), "%i", text variable: Status_GVL.RecipeLine[4].OffsetPattern.Offset_X[5]
    RoundedRectangle (395,58 60x29), "%i", text variable: Status_GVL.RecipeLine[4].OffsetPattern.Offset_X[6]
    RoundedRectangle (466,58 60x29), "%i", text variable: Status_GVL.RecipeLine[4].OffsetPattern.Offset_X[7]
    RoundedRectangle (535,58 60x29), "%i", text variable: Status_GVL.RecipeLine[4].OffsetPattern.Offset_X[8]
    RoundedRectangle (605,59 60x29), "%i", text variable: Status_GVL.RecipeLine[4].OffsetPattern.Offset_X[9]
    RoundedRectangle (674,59 60x29), "%i", text variable: Status_GVL.RecipeLine[4].OffsetPattern.Offset_X[10]
    Label (212,26 25x35), "3"
    Label (280,26 25x35), "4"
    Label (350,26 25x35), "5"
    Label (420,26 25x35), "6"
    Label (488,26 25x35), "7"
    Label (562,26 25x35), "8"
    Label (630,26 25x35), "9"
    Label (700,26 25x35), "10"
    RoundedRectangle (44,96 60x29), "%i", text variable: Status_GVL.RecipeLine[4].OffsetPattern.Offset_Y[1]
    RoundedRectangle (113,96 60x29), "%i", text variable: Status_GVL.RecipeLine[4].OffsetPattern.Offset_Y[2]
    RoundedRectangle (184,96 60x29), "%i", text variable: Status_GVL.RecipeLine[4].OffsetPattern.Offset_Y[3]
    RoundedRectangle (253,96 60x29), "%i", text variable: Status_GVL.RecipeLine[4].OffsetPattern.Offset_Y[4]
    RoundedRectangle (326,95 60x29), "%i", text variable: Status_GVL.RecipeLine[4].OffsetPattern.Offset_Y[5]
    RoundedRectangle (395,95 60x29), "%i", text variable: Status_GVL.RecipeLine[4].OffsetPattern.Offset_Y[6]
    RoundedRectangle (466,95 60x29), "%i", text variable: Status_GVL.RecipeLine[4].OffsetPattern.Offset_Y[7]
    RoundedRectangle (535,95 60x29), "%i", text variable: Status_GVL.RecipeLine[4].OffsetPattern.Offset_Y[8]
    RoundedRectangle (605,96 60x29), "%i", text variable: Status_GVL.RecipeLine[4].OffsetPattern.Offset_Y[9]
    RoundedRectangle (674,96 60x29), "%i", text variable: Status_GVL.RecipeLine[4].OffsetPattern.Offset_Y[10]
    Label (13,162 25x35), "X"
    RoundedRectangle (43,162 60x29), "%i", text variable: Status_GVL.RecipeLine[4].OffsetPattern.Offset_X[13]
    RoundedRectangle (112,162 60x29), "%i", text variable: Status_GVL.RecipeLine[4].OffsetPattern.Offset_X[14]
    RoundedRectangle (183,162 60x29), "%i", text variable: Status_GVL.RecipeLine[4].OffsetPattern.Offset_X[15]
    RoundedRectangle (252,162 60x29), "%i", text variable: Status_GVL.RecipeLine[4].OffsetPattern.Offset_X[16]
    Label (13,201 25x35), "Y"
    RoundedRectangle (325,161 60x29), "%i", text variable: Status_GVL.RecipeLine[4].OffsetPattern.Offset_X[17]
    RoundedRectangle (394,161 60x29), "%i", text variable: Status_GVL.RecipeLine[4].OffsetPattern.Offset_X[18]
    RoundedRectangle (465,161 60x29), "%i", text variable: Status_GVL.RecipeLine[4].OffsetPattern.Offset_X[19]
    RoundedRectangle (534,161 60x29), "%i", text variable: Status_GVL.RecipeLine[4].OffsetPattern.Offset_X[20]
    RoundedRectangle (604,161 60x29), "%i", text variable: Status_GVL.RecipeLine[4].OffsetPattern.Offset_X[21]
    RoundedRectangle (673,161 60x29), "%i", text variable: Status_GVL.RecipeLine[4].OffsetPattern.Offset_X[22]
    RoundedRectangle (43,199 60x29), "%i", text variable: Status_GVL.RecipeLine[4].OffsetPattern.Offset_Y[13]
    RoundedRectangle (112,199 60x29), "%i", text variable: Status_GVL.RecipeLine[4].OffsetPattern.Offset_Y[14]
    RoundedRectangle (183,199 60x29), "%i", text variable: Status_GVL.RecipeLine[4].OffsetPattern.Offset_Y[15]
    RoundedRectangle (252,199 60x29), "%i", text variable: Status_GVL.RecipeLine[4].OffsetPattern.Offset_Y[16]
    RoundedRectangle (325,198 60x29), "%i", text variable: Status_GVL.RecipeLine[4].OffsetPattern.Offset_Y[17]
    RoundedRectangle (394,198 60x29), "%i", text variable: Status_GVL.RecipeLine[4].OffsetPattern.Offset_Y[18]
    RoundedRectangle (465,198 60x29), "%i", text variable: Status_GVL.RecipeLine[4].OffsetPattern.Offset_Y[19]
    RoundedRectangle (534,198 60x29), "%i", text variable: Status_GVL.RecipeLine[4].OffsetPattern.Offset_Y[20]
    RoundedRectangle (604,198 60x29), "%i", text variable: Status_GVL.RecipeLine[4].OffsetPattern.Offset_Y[21]
    RoundedRectangle (673,198 60x29), "%i", text variable: Status_GVL.RecipeLine[4].OffsetPattern.Offset_Y[22]
    Label (69,132 25x35), "13"
    Label (137,132 25x35), "14"
    Label (211,132 25x35), "15"
    Label (279,132 25x35), "16"
    Label (349,132 25x35), "17"
    Label (419,132 25x35), "18"
    Label (487,132 25x35), "19"
    Label (561,132 25x35), "20"
    Label (629,132 25x35), "21"
    Label (699,132 25x35), "22"
    RoundedRectangle (0,262 900x237)
    Label (0,255 900x40), "EDIT OFFSET"
    Label (13,310 25x35), "X"
    RoundedRectangle (43,314 60x29), "%i", text variable: HMI_GVL.arRecipeHMI[4].OffsetPattern.Offset_X[1], input disabled if: Status_GVL.StsEdit[4]
        OnMouseClick: write the text variable via Default
    Label (69,281 25x35), "1"
    RoundedRectangle (112,314 60x29), "%i", text variable: HMI_GVL.arRecipeHMI[4].OffsetPattern.Offset_X[2], input disabled if: Status_GVL.StsEdit[4]
        OnMouseClick: write the text variable via Default
    Label (137,281 25x35), "2"
    RoundedRectangle (183,314 60x29), "%i", text variable: HMI_GVL.arRecipeHMI[4].OffsetPattern.Offset_X[3], input disabled if: Status_GVL.StsEdit[4]
        OnMouseClick: write the text variable via Default
    RoundedRectangle (252,314 60x29), "%i", text variable: HMI_GVL.arRecipeHMI[4].OffsetPattern.Offset_X[4], input disabled if: Status_GVL.StsEdit[4]
        OnMouseClick: write the text variable via Default
    Label (13,349 25x35), "Y"
    RoundedRectangle (325,313 60x29), "%i", text variable: HMI_GVL.arRecipeHMI[4].OffsetPattern.Offset_X[5], input disabled if: Status_GVL.StsEdit[4]
        OnMouseClick: write the text variable via Default
    RoundedRectangle (394,313 60x29), "%i", text variable: HMI_GVL.arRecipeHMI[4].OffsetPattern.Offset_X[6], input disabled if: Status_GVL.StsEdit[4]
        OnMouseClick: write the text variable via Default
    RoundedRectangle (465,313 60x29), "%i", text variable: HMI_GVL.arRecipeHMI[4].OffsetPattern.Offset_X[7], input disabled if: Status_GVL.StsEdit[4]
        OnMouseClick: write the text variable via Default
    RoundedRectangle (534,313 60x29), "%i", text variable: HMI_GVL.arRecipeHMI[4].OffsetPattern.Offset_X[8], input disabled if: Status_GVL.StsEdit[4]
        OnMouseClick: write the text variable via Default
    RoundedRectangle (604,314 60x29), "%i", text variable: HMI_GVL.arRecipeHMI[4].OffsetPattern.Offset_X[9], input disabled if: Status_GVL.StsEdit[4]
        OnMouseClick: write the text variable via Default
    RoundedRectangle (673,314 60x29), "%i", text variable: HMI_GVL.arRecipeHMI[4].OffsetPattern.Offset_X[10], input disabled if: Status_GVL.StsEdit[4]
        OnMouseClick: write the text variable via Default
    Label (211,281 25x35), "3"
    Label (279,281 25x35), "4"
    Label (349,281 25x35), "5"
    Label (419,281 25x35), "6"
    Label (487,281 25x35), "7"
    Label (561,281 25x35), "8"
    Label (629,281 25x35), "9"
    Label (699,281 25x35), "10"
    RoundedRectangle (43,351 60x29), "%i", text variable: HMI_GVL.arRecipeHMI[4].OffsetPattern.Offset_Y[1], input disabled if: Status_GVL.StsEdit[4]
        OnMouseClick: write the text variable via Default
    RoundedRectangle (112,351 60x29), "%i", text variable: HMI_GVL.arRecipeHMI[4].OffsetPattern.Offset_Y[2], input disabled if: Status_GVL.StsEdit[4]
        OnMouseClick: write the text variable via Default
    RoundedRectangle (183,351 60x29), "%i", text variable: HMI_GVL.arRecipeHMI[4].OffsetPattern.Offset_Y[3], input disabled if: Status_GVL.StsEdit[4]
        OnMouseClick: write the text variable via Default
    RoundedRectangle (252,351 60x29), "%i", text variable: HMI_GVL.arRecipeHMI[4].OffsetPattern.Offset_Y[4], input disabled if: Status_GVL.StsEdit[4]
        OnMouseClick: write the text variable via Default
    RoundedRectangle (325,350 60x29), "%i", text variable: HMI_GVL.arRecipeHMI[4].OffsetPattern.Offset_Y[5], input disabled if: Status_GVL.StsEdit[4]
        OnMouseClick: write the text variable via Default
    RoundedRectangle (394,350 60x29), "%i", text variable: HMI_GVL.arRecipeHMI[4].OffsetPattern.Offset_Y[6], input disabled if: Status_GVL.StsEdit[4]
        OnMouseClick: write the text variable via Default
    RoundedRectangle (465,350 60x29), "%i", text variable: HMI_GVL.arRecipeHMI[4].OffsetPattern.Offset_Y[7], input disabled if: Status_GVL.StsEdit[4]
        OnMouseClick: write the text variable via Default
    RoundedRectangle (534,350 60x29), "%i", text variable: HMI_GVL.arRecipeHMI[4].OffsetPattern.Offset_Y[8], input disabled if: Status_GVL.StsEdit[4]
        OnMouseClick: write the text variable via Default
    RoundedRectangle (604,351 60x29), "%i", text variable: HMI_GVL.arRecipeHMI[4].OffsetPattern.Offset_Y[9], input disabled if: Status_GVL.StsEdit[4]
        OnMouseClick: write the text variable via Default
    RoundedRectangle (673,351 60x29), "%i", text variable: HMI_GVL.arRecipeHMI[4].OffsetPattern.Offset_Y[10], input disabled if: Status_GVL.StsEdit[4]
        OnMouseClick: write the text variable via Default
    Label (12,417 25x35), "X"
    RoundedRectangle (42,417 60x29), "%i", text variable: HMI_GVL.arRecipeHMI[4].OffsetPattern.Offset_X[13], input disabled if: Status_GVL.StsEdit[4]
        OnMouseClick: write the text variable via Default
    RoundedRectangle (111,417 60x29), "%i", text variable: HMI_GVL.arRecipeHMI[4].OffsetPattern.Offset_X[14], input disabled if: Status_GVL.StsEdit[4]
        OnMouseClick: write the text variable via Default
    RoundedRectangle (182,417 60x29), "%i", text variable: HMI_GVL.arRecipeHMI[4].OffsetPattern.Offset_X[15], input disabled if: Status_GVL.StsEdit[4]
        OnMouseClick: write the text variable via Default
    RoundedRectangle (251,417 60x29), "%i", text variable: HMI_GVL.arRecipeHMI[4].OffsetPattern.Offset_X[16], input disabled if: Status_GVL.StsEdit[4]
        OnMouseClick: write the text variable via Default
    Label (12,456 25x35), "Y"
    RoundedRectangle (324,416 60x29), "%i", text variable: HMI_GVL.arRecipeHMI[4].OffsetPattern.Offset_X[17], input disabled if: Status_GVL.StsEdit[4]
        OnMouseClick: write the text variable via Default
    RoundedRectangle (393,416 60x29), "%i", text variable: HMI_GVL.arRecipeHMI[4].OffsetPattern.Offset_X[18], input disabled if: Status_GVL.StsEdit[4]
        OnMouseClick: write the text variable via Default
    RoundedRectangle (464,416 60x29), "%i", text variable: HMI_GVL.arRecipeHMI[4].OffsetPattern.Offset_X[19], input disabled if: Status_GVL.StsEdit[4]
        OnMouseClick: write the text variable via Default
    RoundedRectangle (533,416 60x29), "%i", text variable: HMI_GVL.arRecipeHMI[4].OffsetPattern.Offset_X[20], input disabled if: Status_GVL.StsEdit[4]
        OnMouseClick: write the text variable via Default
    RoundedRectangle (603,416 60x29), "%i", text variable: HMI_GVL.arRecipeHMI[4].OffsetPattern.Offset_X[21], input disabled if: Status_GVL.StsEdit[4]
        OnMouseClick: write the text variable via Default
    RoundedRectangle (672,416 60x29), "%i", text variable: HMI_GVL.arRecipeHMI[4].OffsetPattern.Offset_X[22], input disabled if: Status_GVL.StsEdit[4]
        OnMouseClick: write the text variable via Default
    RoundedRectangle (42,454 60x29), "%i", text variable: HMI_GVL.arRecipeHMI[4].OffsetPattern.Offset_Y[13], input disabled if: Status_GVL.StsEdit[4]
        OnMouseClick: write the text variable via Default
    RoundedRectangle (111,454 60x29), "%i", text variable: HMI_GVL.arRecipeHMI[4].OffsetPattern.Offset_Y[14], input disabled if: Status_GVL.StsEdit[4]
        OnMouseClick: write the text variable via Default
    RoundedRectangle (182,454 60x29), "%i", text variable: HMI_GVL.arRecipeHMI[4].OffsetPattern.Offset_Y[15], input disabled if: Status_GVL.StsEdit[4]
        OnMouseClick: write the text variable via Default
    RoundedRectangle (251,454 60x29), "%i", text variable: HMI_GVL.arRecipeHMI[4].OffsetPattern.Offset_Y[16], input disabled if: Status_GVL.StsEdit[4]
        OnMouseClick: write the text variable via Default
    RoundedRectangle (324,453 60x29), "%i", text variable: HMI_GVL.arRecipeHMI[4].OffsetPattern.Offset_Y[17], input disabled if: Status_GVL.StsEdit[4]
        OnMouseClick: write the text variable via Default
    RoundedRectangle (393,453 60x29), "%i", text variable: HMI_GVL.arRecipeHMI[4].OffsetPattern.Offset_Y[18], input disabled if: Status_GVL.StsEdit[4]
        OnMouseClick: write the text variable via Default
    RoundedRectangle (464,453 60x29), "%i", text variable: HMI_GVL.arRecipeHMI[4].OffsetPattern.Offset_Y[19], input disabled if: Status_GVL.StsEdit[4]
        OnMouseClick: write the text variable via Default
    RoundedRectangle (533,453 60x29), "%i", text variable: HMI_GVL.arRecipeHMI[4].OffsetPattern.Offset_Y[20], input disabled if: Status_GVL.StsEdit[4]
        OnMouseClick: write the text variable via Default
    RoundedRectangle (603,453 60x29), "%i", text variable: HMI_GVL.arRecipeHMI[4].OffsetPattern.Offset_Y[21], input disabled if: Status_GVL.StsEdit[4]
        OnMouseClick: write the text variable via Default
    RoundedRectangle (672,453 60x29), "%i", text variable: HMI_GVL.arRecipeHMI[4].OffsetPattern.Offset_Y[22], input disabled if: Status_GVL.StsEdit[4]
        OnMouseClick: write the text variable via Default
    Label (68,387 25x35), "13"
    Label (136,387 25x35), "14"
    Label (210,387 25x35), "15"
    Label (278,387 25x35), "16"
    Label (348,387 25x35), "17"
    Label (418,387 25x35), "18"
    Label (486,387 25x35), "19"
    Label (560,387 25x35), "20"
    Label (628,387 25x35), "21"
    Label (698,387 25x35), "22"
    Button (866,0 35x35), image: VisuSymbols.Symbols.Wrong
        OnMouseClick: CloseDialog Dialog=MOffset_4, Result=OK, NumpadKeypadSet=True
    RoundedRectangle (744,59 60x29), "%i", text variable: Status_GVL.RecipeLine[4].OffsetPattern.Offset_X[11]
    RoundedRectangle (813,59 60x29), "%i", text variable: Status_GVL.RecipeLine[4].OffsetPattern.Offset_X[12]
    Label (769,26 25x35), "11"
    Label (839,26 25x35), "12"
    RoundedRectangle (744,96 60x29), "%i", text variable: Status_GVL.RecipeLine[4].OffsetPattern.Offset_Y[11]
    RoundedRectangle (813,96 60x29), "%i", text variable: Status_GVL.RecipeLine[4].OffsetPattern.Offset_Y[12]
    RoundedRectangle (743,161 60x29), "%i", text variable: Status_GVL.RecipeLine[4].OffsetPattern.Offset_X[23]
    RoundedRectangle (812,161 60x29), "%i", text variable: Status_GVL.RecipeLine[4].OffsetPattern.Offset_X[24]
    RoundedRectangle (743,198 60x29), "%i", text variable: Status_GVL.RecipeLine[4].OffsetPattern.Offset_Y[23]
    RoundedRectangle (812,198 60x29), "%i", text variable: Status_GVL.RecipeLine[4].OffsetPattern.Offset_Y[24]
    Label (768,132 25x35), "23"
    Label (838,132 25x35), "24"
    RoundedRectangle (743,314 60x29), "%i", text variable: HMI_GVL.arRecipeHMI[4].OffsetPattern.Offset_X[11], input disabled if: Status_GVL.StsEdit[4]
        OnMouseClick: write the text variable via Default
    RoundedRectangle (812,314 60x29), "%i", text variable: HMI_GVL.arRecipeHMI[4].OffsetPattern.Offset_X[12], input disabled if: Status_GVL.StsEdit[4]
        OnMouseClick: write the text variable via Default
    Label (768,281 25x35), "11"
    Label (838,281 25x35), "12"
    RoundedRectangle (743,351 60x29), "%i", text variable: HMI_GVL.arRecipeHMI[4].OffsetPattern.Offset_Y[11], input disabled if: Status_GVL.StsEdit[4]
        OnMouseClick: write the text variable via Default
    RoundedRectangle (812,351 60x29), "%i", text variable: HMI_GVL.arRecipeHMI[4].OffsetPattern.Offset_Y[12], input disabled if: Status_GVL.StsEdit[4]
        OnMouseClick: write the text variable via Default
    RoundedRectangle (742,416 60x29), "%i", text variable: HMI_GVL.arRecipeHMI[4].OffsetPattern.Offset_X[23], input disabled if: Status_GVL.StsEdit[4]
        OnMouseClick: write the text variable via Default
    RoundedRectangle (811,416 60x29), "%i", text variable: HMI_GVL.arRecipeHMI[4].OffsetPattern.Offset_X[24], input disabled if: Status_GVL.StsEdit[4]
        OnMouseClick: write the text variable via Default
    RoundedRectangle (742,453 60x29), "%i", text variable: HMI_GVL.arRecipeHMI[4].OffsetPattern.Offset_Y[23], input disabled if: Status_GVL.StsEdit[4]
        OnMouseClick: write the text variable via Default
    RoundedRectangle (811,453 60x29), "%i", text variable: HMI_GVL.arRecipeHMI[4].OffsetPattern.Offset_Y[24], input disabled if: Status_GVL.StsEdit[4]
        OnMouseClick: write the text variable via Default
    Label (767,387 25x35), "23"
    Label (837,387 25x35), "24"
END_VISUALIZATION

// ---- VISUs/Parameter/Recipe/MRecipe.TcVIS
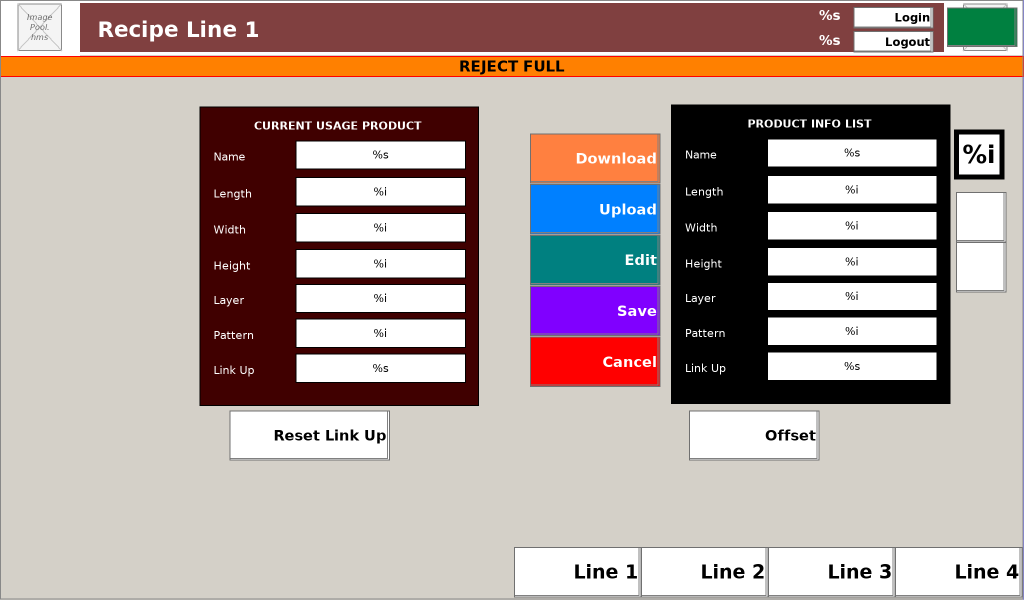
VISUALIZATION MRecipe  // 1024x600
    Frame (0,2 1023x598)
        shows MRecipe_1()
        shows MRecipe_2()
        shows MRecipe_3()
        shows MRecipe_4()
    Button (514,547 127x50), "Line 1", image: VisuSymbols.Symbols.Box
        OnMouseDown: FrameSelectionChange Selection=SelectedFrame=146e207b-fd78-4676-ba16-384fa245d7d2, GlobSel=AssignDir=MainPage.GenElemInst_1003, AssignType=Directly, SelType=Locally
    Button (641,547 127x50), "Line 2", image: VisuSymbols.Symbols.Box
        OnMouseDown: FrameSelectionChange Selection=SelectedFrame=146e207b-fd78-4676-ba16-384fa245d7d2, Selection=1, GlobSel=AssignDir=MainPage.GenElemInst_1003, AssignType=Directly, SelType=Locally
    Button (768,547 127x50), "Line 3", image: VisuSymbols.Symbols.Box
        OnMouseDown: FrameSelectionChange Selection=SelectedFrame=146e207b-fd78-4676-ba16-384fa245d7d2, Selection=2, GlobSel=AssignDir=MainPage.GenElemInst_1003, AssignType=Directly, SelType=Locally
    Button (895,547 127x50), "Line 4", image: VisuSymbols.Symbols.Box
        OnMouseDown: FrameSelectionChange Selection=SelectedFrame=146e207b-fd78-4676-ba16-384fa245d7d2, Selection=3, GlobSel=AssignDir=MainPage.GenElemInst_1003, AssignType=Directly, SelType=Locally
END_VISUALIZATION

// ---- VISUs/Parameter/Recipe/MRecipe_1.TcVIS
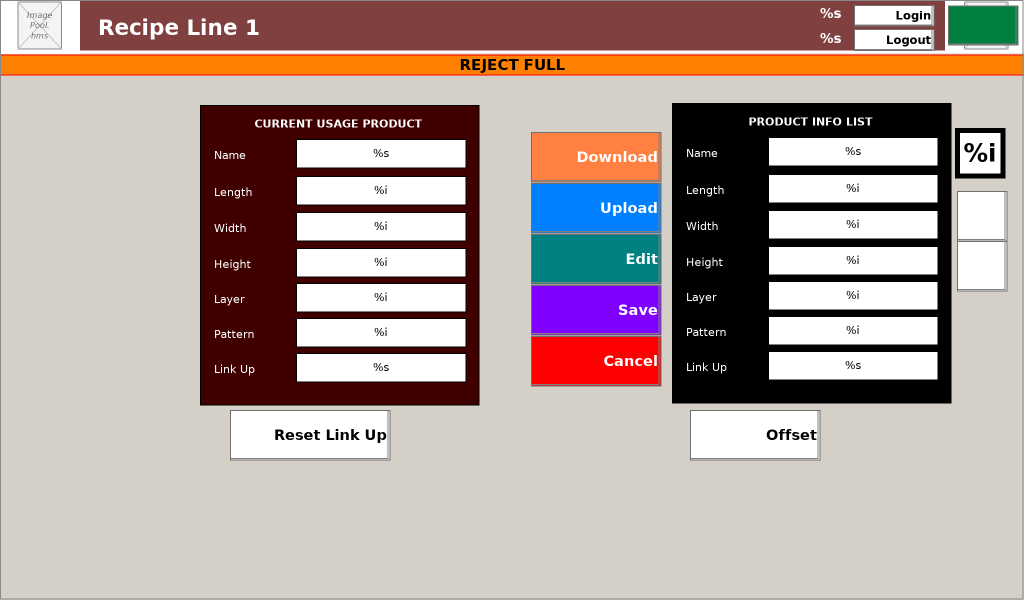
VISUALIZATION MRecipe_1  // 1024x600
    Frame (0,-2 1021x55)
        shows Header()
    Label (95,15 250x25), "Recipe Line 1"
    RoundedRectangle (672,103 279x300)
    Label (697,102 227x40), "PRODUCT INFO LIST"
    Label (683,136 78x35), "Name"
    RoundedRectangle (768,137 170x29), "%s", text variable: HMI_GVL.arRecipeHMI[1].ProductName, input disabled if: Status_GVL.StsEdit[1]
        OnMouseClick: write the text variable via Default
    Label (683,173 78x35), "Length"
    RoundedRectangle (768,174 170x29), "%i", text variable: HMI_GVL.arRecipeHMI[1].ProductLength, input disabled if: Status_GVL.StsEdit[1]
        OnMouseClick: write the text variable via Default
    Label (683,209 78x35), "Width"
    RoundedRectangle (768,210 170x29), "%i", text variable: HMI_GVL.arRecipeHMI[1].ProductWidth, input disabled if: Status_GVL.StsEdit[1]
        OnMouseClick: write the text variable via Default
    Label (683,245 78x35), "Height"
    RoundedRectangle (768,246 170x29), "%i", text variable: HMI_GVL.arRecipeHMI[1].ProductHeight, input disabled if: Status_GVL.StsEdit[1]
        OnMouseClick: write the text variable via Default
    Label (683,280 78x35), "Layer"
    RoundedRectangle (768,281 170x29), "%i", text variable: HMI_GVL.arRecipeHMI[1].Stacking, input disabled if: Status_GVL.StsEdit[1]
        OnMouseClick: write the text variable via Default
    Label (683,315 78x35), "Pattern"
    RoundedRectangle (768,316 170x29), "%i", text variable: HMI_GVL.arRecipeHMI[1].ProductPattern, input disabled if: Status_GVL.StsEdit[1]
        OnMouseClick: write the text variable via Default
    Label (683,350 78x35), "Link Up"
    RoundedRectangle (768,351 170x29), "%s", text variable: HMI_GVL.arRecipeHMI[1].LinkUpSource, input disabled if: Status_GVL.StsEdit[1]
        OnMouseClick: write the text variable via Default
    Button (531,132 130x50), "Download", image: VisuSymbols.Symbols.Download
        tap Status_GVL.Download[1]
    Button (531,183 130x50), "Upload", image: VisuSymbols.Symbols.Eject
        tap Status_GVL.Upload[1]
    Button (531,234 130x50), "Edit", image: VisuSymbols.Symbols.Edit
        tap Status_GVL.Edit[1]
    Button (531,285 130x50), "Save", invisible if: Status_GVL.StsEdit[1], image: VisuSymbols.Symbols.Save
        tap Status_GVL.Save[1]
    Button (531,336 130x50), "Cancel", invisible if: Status_GVL.StsEdit[1], image: VisuSymbols.Symbols.Wrong
        tap Status_GVL.Cancel[1]
    RoundedRectangle (955,128 50x50), "%i", text variable: Status_GVL.RecipeNumber[1]
        OnMouseClick: write Status_GVL.RecipeNumber[1] via Default
    Button (957,191 50x50), image: VisuSymbols.Symbols.TriangleUp
        OnMouseClick: execute {
            IF Status_GVL.StsEdit[1] THEN
            Status_GVL.RecipeNumber[1] := Status_GVL.RecipeNumber[1]+1;
            END_IF
        }
    Button (957,241 50x50), image: VisuSymbols.Symbols.TriangleDown
        OnMouseClick: execute {
            IF Status_GVL.StsEdit[1] THEN
            Status_GVL.RecipeNumber[1] := Status_GVL.RecipeNumber[1]-1;
            END_IF
        }
    Button (690,410 130x50), "Offset", image: VisuSymbols.Symbols.Centered
        OnMouseClick: OpenDialog Dialog=MOffset_1, OpenModal=True, PositionY=0
    Group (200,104 279x356)
        RoundedRectangle (0,1 279x300)
        Label (25,0 227x40), "CURRENT USAGE PRODUCT"
        Label (11,34 78x35), "Name"
        RoundedRectangle (96,35 170x29), "%s", text variable: Status_GVL.RecipeLine[1].ProductName
        Label (11,71 78x35), "Length"
        RoundedRectangle (96,72 170x29), "%i", text variable: Status_GVL.RecipeLine[1].ProductLength
        Label (11,107 78x35), "Width"
        RoundedRectangle (96,108 170x29), "%i", text variable: Status_GVL.RecipeLine[1].ProductWidth
        Label (11,143 78x35), "Height"
        RoundedRectangle (96,144 170x29), "%i", text variable: Status_GVL.RecipeLine[1].ProductHeight
        Label (11,178 78x35), "Layer"
        RoundedRectangle (96,179 170x29), "%i", text variable: Status_GVL.RecipeLine[1].Stacking
        Label (11,213 78x35), "Pattern"
        RoundedRectangle (96,214 170x29), "%i", text variable: Status_GVL.RecipeLine[1].ProductPattern
        Label (11,248 78x35), "Link Up"
        RoundedRectangle (96,249 170x29), "%s", text variable: Status_GVL.RecipeLine[1].LinkUpSource
        Button (30,306 160x50), "Reset Link Up", image: VisuSymbols.Symbols.Eraser
            tap HMI_GVL.Reset_LinkUp[1]
END_VISUALIZATION

